METHOD M_StopCycle
mxStopCycle:= TRUE;
END_METHOD

METHOD M_StopDirect

IF mxCycleBusy THEN
	mxStopDirect:= TRUE;	
END_IF
END_METHOD

METHOD M_StopInit

IF mxInitBusy THEN 
	mxStopInit:= TRUE; 
END_IF
END_METHOD

ACTION Objects:

HydraulicCilinder(
	mxReset:= mxReset,
	mxEmergency:= mxEmergency, 
	mxAutoMode:= mxAutoMode, 
	EndPositionIn:= MachParameters.PositionUpStop,
	EndPositionOut:= ProdParameters.PositionDownStop,
	OffsetPosition:= MachParameters. PositionOffsetZero,
	OffsetAlarmPosition:= MachParameters.PositionOffsetAlarm,
	PositionPhysicalMeasured:=MachParameters.PositionPhyscialMeasured,
	PositionPhysicalMeasuredOld:=MachParameters.PositionPhysicalMeasuredOld,
	PhysicalOffsetPos:=MachParameters.PhysicalOffsetPos,
	RHSR_Blocked:=RHSR_Blocked,
	mxCycleBusy:=mxCycleBusy,
	mxInitBusy:=mxInitBusy,
	mxIsMovingIn=> mxCilIsMovingIn, 
	mxIsMovingOut=> mxCilIsMovingOut,
	ManSpeedCreepIn:=MachParameters.ManSpeedCreep,
	ManSpeedCreepOut:=MachParameters.ManSpeedCreep,
	ManSpeedSlowIn:=MachParameters.ManSpeedSlow,
	ManSpeedSlowOut:=MachParameters.ManSpeedSlow,
	ManSpeedIn:=MachParameters.ManSpeed,
	ManSpeedOut:=MachParameters.ManSpeed,
	mxIsIn=> mxCilIsIn, 
	mxIsOut=> mxCilIsOut,
	Errors=> Errors.HydraulicCilinder);
	
Vacuum(
	mxReset:= mxReset, 
	mxAutoMode:= mxAutoMode);

BlowOff(
	mxReset:= mxReset, 
	mxAutoMode:= mxAutoMode);
END_ACTION

END_FUNCTION_BLOCK

// ---- POUs/InMoldDrying/ProductForming/FB_ProductForming.TcPOU
FUNCTION_BLOCK FB_ProductForming
VAR CONSTANT
	sCycleStateTextDef: ARRAY[0..25]  OF STRING :=	
		['State 0: Wait for Start',
		'State 1: Start wire spray',
		'State 2: Move pond up',
		'State 3: Pond up, await pond up wait time',
		'State 4: Open pulp feeding valve and bubble valve',
		'State 5: Await feeding and bubble time',
		'State 6: Open the vacuum valve and await forming time',
		'State 7: Move pond down',
		'State 8: Start flash spray',
		'State 9: Start after vacuum time and await pre ignition time',
		'State 10: Await after vacuum time done',
		'State 11: Wait for transfer at down position',
		'State 12: Await after blow off time',
		'State 13: ',
		'State 14: ',
		'State 15: ',
		'State 16: ',
		'State 17: ',
		'State 18: ',
		'State 19: ',
		'State 20: Stop cycle state',
		'State 21: Stop direct state'
		];
	
	tCycleStateTimeouts: ARRAY[0..10] OF TIME := 
		[T#10S,T#10S,T#10S,T#10S,T#10S,T#10S,T#10S,T#10S,T#10S,T#10S,
		T#10S];

	sInitStateTextDef: ARRAY[0..10] OF STRING :=
		['State 0: Wait for Start',
		'State 1: Move machinepond down',
		'State 2: Move the spraybar to the rest position',
		'State 3: Description Init State 3',
		'State 4: Description Init State 4',
		'State 5: Description Init State 5',
		'State 6: Description Init State 6',
		'State 7: Description Init State 7',
		'State 8: Description Init State 8',
		'State 9: Description Init State 9',
		'State 10: Stop init state'];

	tInitStateTimeouts: ARRAY[0..10] OF TIME := 
		[T#10S,T#10S,T#10S,T#10S,T#10S,T#10S,T#10S,T#10S,T#10S,T#10S
		,T#10S];
END_VAR

VAR_INPUT
	mxResetCycleState				: BOOL;
	mxResetInitState				: BOOL;
	mxForceInit						: BOOL; (*Reset Calibration Flag*)
	mxReset							: BOOL;	(*Reset Error*)
	mxEmergency						: BOOL;
	mxAutoMode						: BOOL; (* TRUE = Automode *)
	mxStartCycle					: BOOL;
	mxEmptyMachine					: BOOL;
	mxFirstCycle					: BOOL;
	


	
	mxStartTransferMoldVacuum		: BOOL;

	mxAfterBlowOffIsOn				: BOOL;
	ActualPositionTransfermold		: REAL;
	TransfermoldDownPosition		: REAL; // Position at which the transfermold thinks its down.
	TransfermoldMovingDown			: BOOL; // Transfermold is moving down if true.
	TransfermoldMovingUp			: BOOL;
	RHSR_Blocked 					: BOOL;
	
	(*Signals*)
	sgTransferIsDown				: BOOL;(* Reset in cycle *)
	sgAtPosition					: BOOL;
	sgTransferToMoveUp				: BOOL;	
	SgTransferToDownForming			: BOOL; (* Reset at main cycle *)
	
END_VAR
VAR_IN_OUT
	MachParameters					: ST_ProductFormingMachPar;
	SysParameters					: ST_ProductFormingSysPar;
END_VAR
VAR_OUTPUT
(*Errors*)
	Errors							: ST_ProductFormingErrors;
	mxErrorInit						: BOOL;		(* Error, stop immediately. Initialisation neccesary *)
	mxErrorStopinPos				: BOOL;		(* Error, stop in position. Only reset neccesary *)

(* State vars *)
	mxCycleBusy						: BOOL;
	mxInitBusy						: BOOL;
	
(* Vars *)
	mxInitialized					: BOOL;

	mxCilIsMovingIn						: BOOL;
	mxCilIsMovingOut					: BOOL;
	mxCilIsIn							: BOOL;
	mxCilIsOut							: BOOL;

(*Signals*)	
	mxSprayBarAtRestPos					: BOOL;

	
END_VAR
VAR
(* State vars *)
	miCycleState					: INT :=0;
	miCycleOldstate					: INT :=0;
	mxCycleTransitionState			: BOOL := FALSE;
	sCycleStateText					: STRING;
	exCycleTimeOut					: BOOL;		(* Timeout for the whole programcycle *)
	CycleTimeout					: TON;
	CycleTimeOutUpFlank				: R_TRIG;
	mxCycleTimeoutEnable			: BOOL;
	CycleTime						: REAL;
	mxCycleHasError					: BOOL;
	miStopState						: INT;
	mxStopCycle						: BOOL;
	mxStopDirect					: BOOL;
	
	miInitState						: INT	:=0;
	miInitOldstate					: INT	:=0;
	mxInitTransitionState			: BOOL	:= FALSE;
	sInitStateText					: STRING;
	exInitTimeOut					: BOOL;		(* Timeout for the whole programcycle *)
	InitTimeout						: TON;
	InitTimeOutUpFlank				: R_TRIG;
	mxInitTimeoutEnable				: BOOL;
	InitTime						: REAL;
	mxInitHasError					: BOOL;
	mxStartInit						: BOOL;
	mxStopInit						: BOOL;
	
(* Objects *)
(* Forming Mold *)
	MoldVacuum						: FB_MonoValveNoFdbck;							
	MoldBlowOff						: FB_MonoValveNoFdbck;
(* MachinePond *)
	PondHydraulicCilinder			: FB_HydraulicCilinder;
	FeedingPulp						: FB_MonoValve2Fdbck;
(* SprayBar *)	
	WireSprayValve					: FB_MonoValveNoFdbck;
	FlashSprayValve					: FB_MonoValveNoFdbck;
	SprayBarMotor					: FB_NCAxis;	

	(* Interface signals pulp tanks, plup supply*)
	ixPulpTank01					AT %I*: BOOL;
	ixPulpTank02					AT %I*: BOOL;
	ixCssHasAnError					AT %I*: BOOL;
	
	TankLevel01						: FB_AnalogIn4_20mA;
	TankLevel02						: FB_AnalogIn4_20mA;
	
(* Vars *)

	T_PondUpWaitTime	: TON;
	T_FeedingPulp		: TON;
	T_Bubble			: TON;
	
	T_FirstVacuum		: TON;
	T_SecondVacuum		: TON;
	T_ThirdVacuum		: TON;

	T_FormingClosedTime : TON;

	
	FormingVacuumTime	: TIME;
	

	miWireSprayInterval	: INT;
	mxMoveForward		: BOOL;
	miFlashSprayInterval: INT;

	
	RT_ixPulpTank01		: R_TRIG;
	RT_ixPulpTank02		: R_TRIG;
	RT_FlashSprayStarted: R_TRIG;
	RT_InitBusy			: R_TRIG;

	mxPreIgnitionActive	: BOOL;

	mxSprayBarAtRestPosFront: BOOL;
	mxSprayBarAtRestPosBack: BOOL;
	T_SprayDelayTime	: TON;
	T_CycleTimeForKickoffs: TON;
	ActTimeSingleKO		: REAL;
	SR_TanksAreAllmostEmpty: SR;
	mxBubblingReady: BOOL;
	SR_CssHasError: SR;
END_VAR

Error();
Init();
Cycle();
Objects();

mxSprayBarAtRestPos:= mxSprayBarAtRestPosFront OR mxSprayBarAtRestPosBack;
	
mxSprayBarAtRestPosFront := ((SprayBarMotor.ActPosition <= MachParameters.SprayBar.PositionRestFront + 5) AND (SprayBarMotor.ActPosition >= MachParameters.SprayBar.PositionRestFront - 5));
mxSprayBarAtRestPosBack := ((SprayBarMotor.ActPosition <= MachParameters.SprayBar.PositionRestBack + 5) AND (SprayBarMotor.ActPosition >= MachParameters.SprayBar.PositionRestBack - 5));

ACTION Cycle:
(*StateChange (Transition)  Signalgeneration*)
mxCycleTransitionState:=(miCycleState<>miCycleOldstate);
(*State text*)
sCycleStateText:=sCycleStateTextDef[miCycleState];
(*Timeout Watchdog for Statemachine*)
mxCycleTimeoutEnable:=NOT (miCycleState=0) AND NOT mxReset;

CycleTimeout(IN:=mxCycleTimeoutEnable, PT:=tCycleStateTimeouts[miCycleState] );
CycleTimeOutUpFlank(CLK:=CycleTimeout.Q );
miCycleOldstate:=miCycleState;

(*Set Errorbit when Raising edge of Timeout has been detected*)
IF CycleTimeOutUpFlank.Q THEN
	exCycleTimeOut:=TRUE; 			(* 1 Timeout for the whole programcycle *)
END_IF

(*Function to reset the Statemachine*)
IF mxResetCycleState THEN
	mxResetCycleState:= FALSE;
	mxInitialized := FALSE;
	miCycleState:=0;
	miCycleOldstate:=miCycleState;
	mxCycleTransitionState:=FALSE;

	mxStartTransferMoldVacuum:= FALSE;
	mxAfterBlowOffIsOn := FALSE;
	mxStartCycle:= FALSE;
	mxStopCycle:= FALSE;
	mxStopDirect:=FALSE;

	T_FirstVacuum.In := FALSE;
	T_SecondVacuum.IN:= FALSE;
	T_ThirdVacuum.IN := TRUE;
	
	T_PondUpWaitTime.IN:= FALSE;
	T_FeedingPulp.IN:= FALSE;
	T_Bubble.IN:= FALSE;
	
	T_SprayDelayTime.IN:= FALSE;
	T_CycleTimeForKickoffs.IN := FALSE;
	SprayBarMotor.M_Stop();
	
	sgTransferIsDown := FALSE;
	sgAtPosition :=FALSE;
	sgTransferToMoveUp :=FALSE;	
	SgTransferToDownForming :=FALSE; 
END_IF

(*Definition State has Error*)
mxCycleHasError:=FALSE;


(* Set Forming vacuum time when switch over to next pulp tank,
Increase when flah spray is started*)
RT_ixPulpTank01(CLK:= ixPulpTank01);
RT_ixPulpTank02(CLK:= ixPulpTank02);
RT_InitBusy(CLK:= mxInitBusy);
RT_FlashSprayStarted(CLK:= miCycleState = 8);
	
IF RT_ixPulpTank01.Q OR RT_ixPulpTank02.Q OR RT_InitBusy.Q OR TRUE THEN // ----------------------------------------------------------------------------------- TRUE Weghalen wanneer wissel signaal actief
	FormingVacuumTime:= MachParameters.FormingMold.VacuumTime;
ELSIF RT_FlashSprayStarted.Q AND FALSE THEN								// ----------------------------------------------------------------------------------- IDEM voor false.
	IF ixPulpTank01 THEN
		FormingVacuumTime := FormingVacuumTime + (REAL_TO_TIME((TIME_TO_REAL(MachParameters.FormingMold.VacuumTimeIncr ) / 70.0) * (75 -  TankLevel01.EngUnits))); 
	ELSIF ixPulpTank02 THEN
		FormingVacuumTime := FormingVacuumTime + (REAL_TO_TIME((TIME_TO_REAL(MachParameters.FormingMold.VacuumTimeIncr ) / 70.0) * (75 -  TankLevel02.EngUnits))); 
	END_IF
END_IF


// 			Timers			//
T_FeedingPulp(IN:= , PT:= MachParameters.MachinePond.FeedingPulpTime); 
T_Bubble(IN:= , PT:= MachParameters.FormingMold.BubbleTime);
T_FormingClosedTime(IN:= , PT:= MachParameters.FormingMold.ClosedTime);
T_SprayDelayTime(IN:=, PT:=MachParameters.SprayBar.SprayDelayTime);
T_CycleTimeForKickoffs(IN:=, PT:=T#250S);
T_FirstVacuum(IN:= , PT:= FormingVacuumTime);
T_SecondVacuum(IN:= , PT:= MachParameters.FormingMold.SecondVacuum);
T_ThirdVacuum(IN:=, PT:=MachParameters.FormingMold.ThirdVacuum);

// Signal the transfermold that it can start moving down afet T2 has elapsed
IF T_SecondVacuum.Q THEN	
	T_SecondVacuum.IN:= FALSE;
	T_ThirdVacuum.IN := TRUE;
	SgTransferToDownForming:= TRUE; // send transfermold down
END_IF

IF T_ThirdVacuum.Q THEN
	T_ThirdVacuum.IN := FALSE;	
END_IF

// Close feeding pulp valve after timer is done
IF T_FeedingPulp.Q THEN 
	T_FeedingPulp.IN := FALSE;
	FeedingPulp.M_Close(); 
END_IF
			
(*Cycle State's*)
CASE miCycleState OF

{region "Steps overview"}	
	(*
	-Start wire spray
	-move pond up
	-Open blow off valve (bubble) 
	-Await bubble time
	-Close feeding valve/blow off valve/start vacuum + timer
	-Wait for vacuum timer
	-move pond down
	-Start flash spray
	-Start after vacuum timer/Pre-ignition timer
	-After vacuum time is done, -> Move down to Transfer Mold
	-Wait for transfer down 	<- from transfer mold
	-Open blow off valve
	-Start forming timer
	-Start blow off timer
	-Signal to transfer 		-> Move up to transfer mold
	-Wait for start forming (start cycle)		<- from transfer mold
	*)
{endregion}
	0:
		IF mxStopDirect THEN
			mxStopDirect:= FALSE;
			miCycleState:= 21;
		ELSIF mxStopCycle AND mxEmptyMachine THEN
			mxEmptyMachine:= FALSE;
			T_CycleTimeForKickoffs.IN := FALSE;	// Start timer to measure the cycle time of the transfer mold.
			miCycleState:= 0;
		ELSIF mxStopCycle THEN
			mxStopCycle:= FALSE;
			miStopState:= miCycleState;
			miCycleState:= 20;
		ELSIF mxStartCycle THEN
			mxStartCycle:= FALSE;
			T_CycleTimeForKickoffs.IN := TRUE;	// Start timer to measure the cycle time of the transfer mold.
			mxStartTransferMoldVacuum:= FALSE;
			
			mxMoveForward:= FALSE;				(* Check if at rest back position, then move forward, else move backward *)
			IF SprayBarMotor.ActPosition < MachParameters.SprayBar.PositionRestBack + 5 AND SprayBarMotor.ActPosition > MachParameters.SprayBar.PositionRestBack - 5 THEN
				mxMoveForward:= TRUE;
			END_IF	
			(* If parameter = 0 then do not perform spray, if 1 then always perform spray, other: perform every x time *)
			IF MachParameters.SprayBar.WireSprayInterval > 0 AND ((miWireSprayInterval = MachParameters.SprayBar.WireSprayInterval) OR MachParameters.SprayBar.WireSprayInterval = 1) THEN
				miWireSprayInterval:= miWireSprayInterval - 1;		
				miCycleState:= 1;
			ELSE
				miWireSprayInterval:= miWireSprayInterval - 1;
				miCycleState:=2 ;
			END_IF
			IF miWireSprayInterval <=0 THEN miWireSprayInterval:= MachParameters.SprayBar.WireSprayInterval; END_IF		//Write to par if is lower then 0
		END_IF
		
	
	1: // Start Wire Spray 
		IF mxMoveForward THEN
			IF SprayBarMotor.ActPosition >= MachParameters.SprayBar.PositionStartWireFwd THEN
				WireSprayValve.M_On();
			END_IF
			IF SprayBarMotor.ActPosition >= MachParameters.SprayBar.PositionStopWireFwd THEN
				WireSprayValve.M_Off();
			END_IF
		ELSE
			IF SprayBarMotor.ActPosition <= MachParameters.SprayBar.PositionStartWireBkw THEN
				WireSprayValve.M_On();
			END_IF
			IF SprayBarMotor.ActPosition <= MachParameters.SprayBar.PositionStopWireBkw THEN
				WireSprayValve.M_Off();
			END_IF
		END_IF
			
		IF mxStopDirect THEN
			mxStopDirect:= FALSE;
			miCycleState:= 21;
		ELSIF mxStopCycle THEN
			mxStopCycle:= FALSE;			
			miStopState:= miCycleState;
			miCycleState:= 20;
		ELSIF mxMoveForward  THEN
			IF SprayBarMotor.M_MoveAbsolute(Velocity:= MachParameters.SprayBar.AutoVelocity, Position:= MachParameters.SprayBar.PositionRestFront) THEN
				miCycleState:= 2;	
			END_IF
		ELSIF NOT mxMoveForward THEN
			IF SprayBarMotor.M_MoveAbsolute(Velocity:= MachParameters.SprayBar.AutoVelocity, Position:= MachParameters.SprayBar.PositionRestBack) THEN
				miCycleState:= 2;	
			END_IF
		END_IF
	
	2:	// Move pond up
		IF (PondHydraulicCilinder.ActPosition > (MachParameters.MachinePond.PositionUpStop - MachParameters.MachinePond.BubblingPositionOffset)) THEN
			IF MoldBlowOff.M_On() THEN T_Bubble.IN:= TRUE; END_IF  // When the machine pond is almost up -> Start bubbling (open valve)
		END_IF
	
		IF mxStopDirect THEN
			mxStopDirect:= FALSE;
			miCycleState:= 21;
		ELSIF mxStopCycle THEN
			mxStopCycle:= FALSE;
			PondHydraulicCilinder.M_Stop();		
			miStopState:= miCycleState;
			miCycleState:= 20;
		ELSIF PondHydraulicCilinder.M_Move(End_Position:= MachParameters.MachinePond.PositionUpStop, Slow_Position:= MachParameters.MachinePond.PositionUpSlow) THEN
			miCycleState:= 3;
		END_IF
	
	3:	// pulp supply open when bubbling is done.		
		IF mxStopDirect THEN
			mxStopDirect:= FALSE;
			miCycleState:= 21;
		ELSIF mxStopCycle THEN
			mxStopCycle:= FALSE;
			miStopState:= miCycleState;
			miCycleState:= 20;	
		ELSIF T_Bubble.Q OR TRUE THEN // REMOVE TRUE when done with testing.
			T_Bubble.IN := FALSE;
			MoldBlowOff.M_Off();	
		
			// open feeding valve
			FeedingPulp.M_Open();  
			T_FeedingPulp.IN:= TRUE;
			
			//Start first vacuum
			MoldVacuum.M_On();	// open the vacuum valve and start first vac. timer.
			T_FirstVacuum.IN := TRUE;	
			
			miCycleState:= 4;
		END_IF	
		
	4:	// First vacuum time is finished, start 2nd vacuum time	
		IF mxStopDirect THEN
			mxStopDirect:= FALSE;
			miCycleState:= 21;
		ELSIF mxStopCycle THEN
			mxStopCycle:= FALSE;
			miStopState:= miCycleState;
			miCycleState:= 20;	
		ELSIF T_FirstVacuum.Q THEN
			T_FirstVacuum.IN := FALSE;
			T_SecondVacuum.IN := TRUE;	
			miCycleState:= 5;
		END_IF		
	
	5:	///When first vacuum is finished and 2nd started, move pond down.
		IF mxStopDirect THEN
			mxStopDirect:= FALSE;
			miCycleState:= 21;
		ELSIF mxStopCycle THEN
			mxStopCycle:= FALSE;		
			miStopState:= miCycleState;
			miCycleState:= 20;
		ELSIF PondHydraulicCilinder.M_Move(End_Position:= MachParameters.MachinePond.PositionDownStop, Slow_Position:= MachParameters.MachinePond.PositionDownSlow) THEN
			T_SprayDelayTime.IN:= TRUE;		
			
			IF T_SprayDelayTime.Q THEN
				T_SprayDelayTime.IN :=FALSE;	
			
				mxMoveForward:= FALSE;
				IF SprayBarMotor.ActPosition < MachParameters.SprayBar.PositionRestBack + 5 AND SprayBarMotor.ActPosition > MachParameters.SprayBar.PositionRestBack - 5 THEN
					mxMoveForward:= TRUE;
				END_IF	
				
				(* If parameter = 0 then do not perform spray, if 1 then always perform spray, other: perform every x time *)
				IF MachParameters.SprayBar.FlashSprayInterval > 0 AND ((miFlashSprayInterval = MachParameters.SprayBar.FlashSprayInterval) OR MachParameters.SprayBar.FlashSprayInterval = 1) THEN
					miFlashSprayInterval:= miFlashSprayInterval - 1;
					miCycleState:= 6; 
				ELSE
					miFlashSprayInterval:= miFlashSprayInterval - 1;		
					miCycleState:= 7;
				END_IF
				IF miFlashSprayInterval <=0 THEN miFlashSprayInterval:= MachParameters.SprayBar.FlashSprayInterval; END_IF 	// Write to par if is lower then 0
			END_IF
		END_IF
	
	6: 	// Start flash spray 
		IF mxMoveForward THEN
			IF SprayBarMotor.ActPosition >= MachParameters.SprayBar.PositionStartFlashFwd THEN
				FlashSprayValve.M_On();
			END_IF
			IF SprayBarMotor.ActPosition >= MachParameters.SprayBar.PositionStopFlashFwd THEN
				FlashSprayValve.M_Off();
			END_IF
		ELSE
			IF SprayBarMotor.ActPosition <= MachParameters.SprayBar.PositionStartFlashBkw THEN
				FlashSprayValve.M_On();
			END_IF
			IF SprayBarMotor.ActPosition <= MachParameters.SprayBar.PositionStopFlashBkw THEN
				FlashSprayValve.M_Off();
			END_IF
		END_IF

		IF mxStopDirect THEN
			mxStopDirect:= FALSE;
			miCycleState:= 21;
		ELSIF mxStopCycle THEN
			mxStopCycle:= FALSE;
			miStopState:= miCycleState;
			miCycleState:= 20;
		ELSIF mxMoveForward THEN
			IF SprayBarMotor.M_MoveAbsolute(Velocity:= MachParameters.SprayBar.AutoVelocity, Position:= MachParameters.SprayBar.PositionRestFront) THEN
				miCycleState:= 7;	
			END_IF
		ELSIF NOT mxMoveForward THEN
			IF SprayBarMotor.M_MoveAbsolute(Velocity:= MachParameters.SprayBar.AutoVelocity, Position:= MachParameters.SprayBar.PositionRestBack) THEN
				miCycleState:= 7;	
			END_IF
		END_IF

	7:	// Close forming mold vacuum valve on the way down of transfermold.
		IF TransfermoldMovingDown AND (ActualPositionTransfermold < (TransfermoldDownPosition + MachParameters.FormingMold.StopVacuumAtTrPosOffset)) THEN
			T_ThirdVacuum.IN := FALSE; // Abort third vacuum timer, to indicate total time.				
			MoldVacuum.M_Off();
		END_IF
		
		IF TransfermoldMovingDown AND (ActualPositionTransfermold < (TransfermoldDownPosition + MachParameters.FormingMold.StartBlowOffAtTrPosOffset)) THEN				
			MoldBlowoff.M_On();
		END_IF

		IF mxStopDirect THEN
			mxStopDirect:= FALSE;
			miCycleState:= 21;
		ELSIF mxStopCycle THEN
			mxStopCycle:= FALSE;
			miStopState:= miCycleState;
			miCycleState:= 20;
		ELSIF sgTransferIsDown THEN
			sgTransferIsDown:= FALSE;
			miCycleState:= 8;
		END_IF
		
	8:	// Close time (time the transfer is closed on the formingmold).
		T_FormingClosedTime.IN:= TRUE;

		IF mxStopDirect THEN
			mxStopDirect:= FALSE;
			miCycleState:= 21;
		ELSIF mxStopCycle THEN
			mxStopCycle:= FALSE;
			miStopState:= miCycleState;
			miCycleState:= 20;
		ELSIF T_FormingClosedTime.Q THEN	// Signal main cycle that transfer to start moving up again.
			T_FormingClosedTime.In:= FALSE;
			sgTransferToMoveUp:=TRUE;
			miCycleState:= 9;
		END_IF

	
	9:	// Switch blowoff due to transfer position 
	//	IF TransfermoldMovingUp AND 
	//	(ActualPositionTransfermold > (TransfermoldDownPosition + MachParameters.FormingMold.StartBlowOffAtTrPosOffset)) THEN				
	//		MoldBlowoff.M_On();
	//	END_IF

		IF mxStopDirect THEN
			mxStopDirect:= FALSE;
			miCycleState:= 21;
		ELSIF mxStopCycle THEN
			mxStopCycle:= FALSE;
			miStopState:= miCycleState;
			miCycleState:= 20;
		ELSIF TransfermoldMovingUp AND 
		(ActualPositionTransfermold > (TransfermoldDownPosition + MachParameters.FormingMold.StopBlowOffAtTrPosOffset)) THEN				
			MoldBlowoff.M_Off();
			
			ActTimeSingleKO := TIME_TO_REAL(T_CycleTimeForKickOffs.ET);
			T_CycleTimeForKickoffs.IN := FALSE;
			miCycleState:= 0;
		END_IF
		
	(* Stop Cycle *)
	20:
		FeedingPulp.M_Close();				// on controlled stop, close the pulpfeeding valve to prevent flooding.
	
		IF mxStopDirect THEN
			mxStopDirect:= FALSE;
			miCycleState:= 21;
		ELSIF mxStartCycle THEN
			mxStartCycle:= FALSE;
			miCycleState:= miStopState;
			T_CycleTimeForKickoffs.IN := FALSE;	
		END_IF
	
	(* Stop Direct*)
	21:
		T_PondUpWaitTime.IN:= FALSE;
		T_FeedingPulp.IN:= FALSE;
		T_Bubble.IN:= FALSE;
		
		T_FirstVacuum.IN:= FALSE;
		T_SecondVacuum.IN:= FALSE;
		T_ThirdVacuum.IN := FALSE;
		
		T_CycleTimeForKickoffs.IN := FALSE;	// Start timer to measure the cycle time of the transfer mold.
		ActTimeSingleKO := 0;
		
	(* Forming Mold *)
		MoldVacuum.M_Off();				
		MoldBlowOff.M_Off();
	(* MachinePond *)
		PondHydraulicCilinder.M_StopDirect();
		FeedingPulp.M_Close();
	(* SprayBar *)	
		WireSprayValve.M_Off();
		FlashSprayValve.M_Off();
		SprayBarMotor.M_Stop();

		mxStartCycle:= FALSE;
		mxStopCycle:= FALSE;
		mxStopDirect:=FALSE;
		mxInitialized:= FALSE;

		sgTransferIsDown := FALSE;
		sgAtPosition :=FALSE;
		sgTransferToMoveUp :=FALSE;	
		SgTransferToDownForming :=FALSE; 
		
		miCycleState:= 0;

END_CASE

mxCycleBusy:= miCycleState<>0 AND NOT (miCycleState=20);
END_ACTION

ACTION Error:
SR_TanksAreAllmostEmpty(SET1:=(TankLevel01.EngUnits < 5) AND (TankLevel02.EngUnits < 5), RESET:=mxReset, Q1=>Errors.LowLvlOnBothTanks);  
SR_CssHasError(SET1:=ixCssHasAnError, Reset:=mxReset, Q1=>Errors.CssHasError);



(*************************************************************************************************)
mxErrorInit:= Errors.HydraulicPump.Thermal;
mxErrorStopinPos:= FALSE;
END_ACTION

ACTION Init:
(*StateChange (Transition)  Signalgeneration*)
mxInitTransitionState:=(miInitState<>miInitOldstate);
(*State text*)
sInitStateText:=sInitStateTextDef[miInitState];
(*Timeout Watchdog for Statemachine*)
mxInitTimeoutEnable:=NOT (miInitState=0)  AND NOT mxReset;

InitTimeout(IN:=mxInitTimeoutEnable  , PT:=tInitStateTimeouts[miInitState] );
InitTimeOutUpFlank(CLK:=InitTimeout.Q );
miInitOldstate:=miInitState;

(*Set Errorbit when Raising edge of Timeout has been detected*)
IF InitTimeOutUpFlank.Q THEN
	exInitTimeOut:=TRUE; 			(* 1 Timeout for the whole programcycle *)
END_IF

(*Function to reset the Statemachine*)
IF mxResetInitState THEN
	mxResetInitState:=FALSE;
	mxInitialized:= FALSE;
	miInitState:=0;
	miInitOldstate:=miInitState;
	mxInitTransitionState:=FALSE;
	
	mxStartInit:= FALSE;
	mxStopInit:= FALSE;
END_IF

(*Definition State has Error*)
mxInitHasError:=FALSE;

CASE miInitState OF
	0:
		IF mxStartInit THEN
			mxStartInit:= FALSE;
			mxInitialized:= FALSE;

		(* Forming Mold *)
			MoldVacuum.M_Off();				
			MoldBlowOff.M_Off();
		(* MachinePond *)
			FeedingPulp.M_Close();
		(* SprayBar *)	
			WireSprayValve.M_Off();
			FlashSprayValve.M_Off();
			(* AT init write intervals *)
			miWireSprayInterval:= MachParameters.SprayBar.WireSprayInterval;
			miFlashSprayInterval:= MachParameters.SprayBar.FlashSprayInterval;
			
			miInitState:= 1;
		END_IF

	(* Move Pond down *)	
	1:
		IF mxStopInit THEN
			mxStopInit:= FALSE;
			
			miInitState:= 10;			
		ELSIF PondHydraulicCilinder.M_Move(End_Position:= MachParameters.MachinePond.PositionDownStop, Slow_Position:= MachParameters.MachinePond.PositionDownSlow) THEN
			
			miInitState:= 2;
		END_IF				

	(* Move spraybar to rest position *)	
	2:
		IF mxStopInit THEN
			mxStopInit:= FALSE;
			
			miInitState:= 10;			
		ELSIF SprayBarMotor.M_MoveAbsolute(Position:= MachParameters.SprayBar.PositionRestBack, Velocity:= MachParameters.SprayBar.AutoVelocity) THEN
			mxInitialized:= TRUE;
			
			// stop the pump en cylinder of the pond
			PondHydraulicCilinder.M_Stop();
			
			miInitState:= 0;
		END_IF

	10:
		PondHydraulicCilinder.M_Stop();
		SprayBarMotor.M_Stop();

		mxStartInit:= FALSE;
		mxStopInit:= FALSE;
		mxInitialized:= FALSE;
		
		miInitState:= 0;
END_CASE

mxInitBusy:= miInitState<>0;
END_ACTION

METHOD M_EmptyMachine

IF mxCycleBusy THEN
	mxEmptyMachine:= TRUE;	
END_IF
END_METHOD

METHOD M_StartCycle

IF NOT mxCycleBusy THEN
	mxStartCycle:= TRUE;
	mxStopCycle:=False;
END_IF
END_METHOD

METHOD M_StartInit

IF NOT mxInitBusy THEN 
	mxStartInit:= TRUE;
END_IF
END_METHOD

METHOD M_StopCycle

IF mxCycleBusy THEN
	mxStopCycle:= TRUE;
END_IF
END_METHOD

METHOD M_StopDirect

IF mxCycleBusy THEN
	mxStopDirect:= TRUE;	
END_IF
END_METHOD

METHOD M_StopInit

IF mxInitBusy THEN 
	mxStopInit:= TRUE; 
END_IF
END_METHOD

ACTION Objects:

MoldVacuum(
	mxReset:= mxReset,
	mxAutoMode:= mxAutoMode,
	mxEmergency:= mxEmergency);

MoldBlowOff(
	mxReset:= mxReset,
	mxAutoMode:= mxAutoMode,
	mxEmergency:= mxEmergency);
	
PondHydraulicCilinder(
	mxReset:= mxReset,
	mxAutoMode:= mxAutoMode,
	mxEmergency:= mxEmergency,
	EndPositionIn:= MachParameters.MachinePond.PositionDownStop,
	EndPositionOut:= MachParameters.MachinePond.PositionUpStop,
	OffsetPosition:= MachParameters.MachinePond.PositionOffsetZero,
	OffsetAlarmPosition:= MachParameters.MachinePond.PositionOffsetAlarm,
	PositionPhysicalMeasured:=MachParameters.MachinePond.PositionPhyscialMeasured,
	PositionPhysicalMeasuredOld:=MachParameters.MachinePond.PositionPhysicalMeasuredOld,
	PhysicalOffsetPos:=MachParameters.MachinePond.PhysicalOffsetPos,
	RHSR_Blocked := RHSR_Blocked,
	SlowValveIsInverted := FALSE,
	mxIsVertical := TRUE,
	mxIsMovingIn=> mxCilIsMovingIn, 
	mxIsMovingOut=> mxCilIsMovingOut, 
	mxIsIn=> mxCilIsIn, 
	mxIsOut=> mxCilIsOut,
	Errors=> );


FeedingPulp(
	mxReset:= mxReset,
	mxAutoMode:= mxAutoMode,
	mxEmergency:= mxEmergency,
	MachParameters:= MachParameters.MachinePond.FeedingPulp);

WireSprayValve(
	mxReset:= mxReset,
	mxAutoMode:= mxAutoMode,
	mxEmergency:= mxEmergency);

FlashSprayValve(
	mxReset:= mxReset,
	mxAutoMode:= mxAutoMode,
	mxEmergency:= mxEmergency);

SprayBarMotor(
	mxEnable:= NOT mxEmergency, 
	mxInhibit:=FALSE , 
	mxAutoMode:= mxAutoMode, 
	mxReset:= mxreset, 
	mxEmergency:= mxEmergency, 
	mxSimulation:= , 
	mxFirstCycle:= mxFirstCycle, 
	mxResetCycle:= , 
	mxDisable_Positive:=FALSE , 
	mxDisable_Negative:=FALSE , 
	mxBlockHMI:=FALSE , 
	mrOverride:= 100,
	mrHomePos:=MachParameters.SprayBar.PositionHome,
	mrVelocityManual:= MachParameters.SprayBar.ManualVelocity, 
	SysParameters:= SysParameters.SprayBar, 
	mxCycleBusy=> , 
	mxRunning=> , 
	Errors=> errors.SprayBar.NCAxisError, 
	Error=> , 
	ErrorStop=> , 
	axStatus=> , 
	ActPosition=> , 
	ActVelocity=> , 
	axAxis=> );
	
TankLevel01(
	EngLowLimit:= 0, 
	EngUpperLimit:= 100, 
	maOut=> , 
	EngUnits=> , 
	EngFilt=> , 
	OverRange=> , 
	UnderRange=> );
	
TankLevel02(
	EngLowLimit:= 0, 
	EngUpperLimit:= 100, 
	maOut=> , 
	EngUnits=> , 
	EngFilt=> , 
	OverRange=> , 
	UnderRange=> );
END_ACTION

END_FUNCTION_BLOCK

// ---- POUs/Standard/HydraulicCilinder/FB_HydraulicCilinder.TcPOU
FUNCTION_BLOCK FB_HydraulicCilinder

VAR_INPUT

	mxReset							: BOOL;	(*Reset Error*)
	mxEmergency						: BOOL;
	mxAutoMode						: BOOL; (* TRUE = Automode *)
	EndPositionIn					: REAL;
	EndPositionOut					: REAL;
	OffsetPosition					: REAL;
	OffsetAlarmPosition				: REAL;	
	PositionPhysicalMeasured		: REAL;	
	RHSR_Blocked					: BOOL; (*IF true, then movement of the cylinder is blocked by the red hot safetyrules.*)
	SlowValveIsInverted				: BOOL;
	mxIsVertical					: BOOL;
	
		// used in M_move
	mxMoveIn						: BOOL;
	mxMoveOut						: BOOL;
	
END_VAR
VAR_OUTPUT
(*Errors*)
	Errors							: ST_HydraulicErrors;
	mxErrorInit						: BOOL;		(* Error, stop immediately. Initialisation neccesary *)
	mxErrorStopinPos				: BOOL;		(* Error, stop in position. Only reset neccesary *)

(* State vars *)
	mxCycleBusy						: BOOL;
	mxInitBusy						: BOOL;
	
(* Vars *)
	mxInitialized					: BOOL;
	ActPosition						: REAL;
	ActMeasuredPosition				: REAL;
	mxSlowActive					: BOOL;
	mxIsMovingIn					: BOOL;
	mxIsMovingOut					: BOOL;
	mxIsIn							: BOOL;
	mxIsOut							: BOOL;
END_VAR
VAR
(* State vars *)
	miCycleState					: INT :=0;
	miCycleOldstate					: INT :=0;
	mxCycleTransitionState			: BOOL := FALSE;
	sCycleStateText					: STRING;
	exCycleTimeOut					: BOOL;		(* Timeout for the whole programcycle *)
	CycleTimeout					: TON;
	CycleTimeOutUpFlank				: R_TRIG;
	mxCycleTimeoutEnable			: BOOL;
	CycleTime						: REAL;
	mxCycleHasError					: BOOL;
	miStopState						: INT;
	mxStartCycle					: BOOL;
	mxStopCycle						: BOOL;
	mxStopDirect					: BOOL;
	
	miInitState						: INT	:=0;
	miInitOldstate					: INT	:=0;
	mxInitTransitionState			: BOOL	:= FALSE;
	sInitStateText					: STRING;
	exInitTimeOut					: BOOL;		(* Timeout for the whole programcycle *)
	InitTimeout						: TON;
	InitTimeOutUpFlank				: R_TRIG;
	mxInitTimeoutEnable				: BOOL;
	InitTime						: REAL;
	mxInitHasError					: BOOL;
	mxStartInit						: BOOL;
	mxStopInit						: BOOL;

	(* Objects *)
	HydraulicIn						: FB_MonoValveNoFdbck;
	HydraulicOut					: FB_MonoValveNoFdbck;
	HydraulicSlow					: FB_MonoValveNoFdbck;
	HydraulicPos 					: FB_BalluffPosition;

	RodSidePressure					: FB_AnalogIn4_20mA;
	BottomSidePressure				: FB_AnalogIn4_20mA;
	
	EndPosition						: REAL; (* Destination position *)
	SlowPosition					: REAL; (* Slow position *)

	FT_ValveInOff					: F_TRIG;
	FT_ValveOutOff					: F_TRIG;
	HydraulicStoredPosition			: REAL;
	

	
	Hysteresis: REAL := 1;
	mxMoveReadyWithoutMoving: BOOL;
	
	RT_Emergency: R_Trig;
	FT_AutoMode: F_TRIG;
END_VAR
VAR_IN_OUT
	PositionPhysicalMeasuredOld		: REAL;
	PhysicalOffsetPos				: REAL;
END_VAR

Error();
Objects();

RT_Emergency(CLK:= mxEmergency);
FT_AutoMode(CLK:=mxAutoMode);

Hysteresis := 3;

// Calculate correction on actual balluf position to a virtual "zero" position.
IF PositionPhysicalMeasured <> PositionPhysicalMeasuredOld THEN
	PhysicalOffsetPos := (HydraulicPos.Position- (OffsetPosition + PositionPhysicalMeasured));
END_IF

// Create a virtual zero position by substracting a calculated offset
ActPosition:= HydraulicPos.Position - PhysicalOffsetPos;
ActMeasuredPosition:= HydraulicPos.Position;

mxIsMovingIn:= HydraulicIn.mxIsOn;
mxIsMovingOut:= HydraulicOut.mxIsOn;

mxIsIn:= (ActPosition <= (EndPositionIn + Hysteresis)) AND (ActPosition >= (EndPositionIn - Hysteresis));
mxIsOut:= (ActPosition <= (EndPositionOut + Hysteresis)) AND (ActPosition >= (EndPositionOut - Hysteresis));

(*Overwrite previous value*)
PositionPhysicalMeasuredOld := PositionPhysicalMeasured;

(* Used for sending slow settings to flow/pressure *) 
mxSlowActive:= HydraulicSlow.mxIsOn;


// Close valves on emergency stop.
IF RT_Emergency.Q OR FT_AutoMode.Q THEN
	HydraulicSlow.M_Off();
	HydraulicIn.M_Off();
	HydraulicOut.M_Off();
END_IF

ACTION Error:
Errors.BallufError:= HydraulicPos.Error;

(* When out of range up/down position *)

	IF (mxIsVertical AND (ActPosition > (EndPositionIn + OffsetAlarmPosition) OR ActPosition < (EndPositionOut - OffsetAlarmPosition))) OR 
		(NOT mxIsVertical AND (ActPosition < (EndPositionIn - OffsetAlarmPosition) OR ActPosition > (EndPositionOut + OffsetAlarmPosition))) THEN
		Errors.PositionError:= TRUE;
	ELSIF mxReset THEN
		Errors.PositionError:= FALSE;
	END_IF

(* Als valve up/down uit gaat, positie opslaan en controleren of deze veranderd tov de act positie*)
FT_ValveInOff(CLK:= HydraulicIn.mxIsOn);
FT_ValveOutOff(CLK:= HydraulicOut.mxIsOn);
IF FT_ValveInOff.Q OR FT_ValveOutOff.Q THEN HydraulicStoredPosition:= ActPosition; END_IF
IF mxReset THEN
	HydraulicStoredPosition:= ActPosition;
	Errors.IsMovingWithoutActivation:= FALSE;
ELSIF NOT HydraulicIn.mxIsOn AND NOT HydraulicOut.mxIsOn AND ((HydraulicStoredPosition > (ActPosition + 10)) OR (HydraulicStoredPosition < (ActPosition - 10))) THEN
	Errors.IsMovingWithoutActivation:= TRUE;
END_IF

(***************************************************************************************)
mxErrorStopInPos:= Errors.PositionError OR Errors.IsMovingWithoutActivation;
mxErrorInit:= FALSE;
END_ACTION

METHOD M_Move : BOOL
VAR_INPUT
	End_Position		: REAL; (* Destination position *)
	Slow_Position		: REAL; (* Slow position *)
END_VAR
VAR_OUTPUT
END_VAR
VAR


	mxMoveINReady: BOOL;
	mxMoveOutReady: BOOL;


END_VAR
(* Pass through parameters *) 
EndPosition:= End_Position;
SlowPosition:= Slow_Position;


mxMoveReadyWithoutMoving := FALSE;

(* bv atc pos = 0, end = 100  *)
IF (mxIsVertical AND (ActPosition <= (EndPosition - Hysteresis)) AND NOT mxMoveOut) OR			// Vertical movement (up)
	(NOT mxIsVertical AND (ActPosition >= (EndPosition + Hysteresis))  AND NOT mxMoveOut) THEN		// Horizontal movement (in)
	mxMoveIn:= TRUE;
	MxMoveOut:= FALSE;
	HydraulicIn.M_On();
	HydraulicOut.M_Off(); 	
ELSIF (mxIsVertical AND (ActPosition >= (EndPosition + Hysteresis)) AND NOT mxMoveIn) OR 			// Vertical movement (down)
	(NOT mxIsVertical AND (ActPosition <= (EndPosition - Hysteresis)) AND NOT mxMoveIn) THEN		// Horizontal movement (out)
	mxMoveIn:= FALSE;
	MxMoveOut:= TRUE;
	HydraulicIn.M_Off();
	HydraulicOut.M_On(); 
ELSE
	mxMoveReadyWithoutMoving:=TRUE;
END_IF

(* Move in *)	
IF mxMoveIn THEN
	IF (mxIsVertical AND (ActPosition > SlowPosition)) OR 				// Vertical movement
		(NOT mxIsVertical AND (ActPosition < SlowPosition))	THEN 		// Horizontal movement.
		HydraulicSlow.M_On();
	END_IF
END_IF

(* Move out *)
IF mxMoveOut THEN
	IF (mxIsVertical AND (ActPosition < SlowPosition)) OR 				// Vertical movement
	(NOT mxIsVertical AND (ActPosition > SlowPosition)) THEN			// Horizontal movement
		HydraulicSlow.M_On();
	END_IF
END_IF

mxMoveInReady := (mxMoveIn AND ((ActPosition >= (EndPosition - Hysteresis)) AND (ActPosition <= (EndPosition + Hysteresis))));
mxMoveOutReady := (mxMoveOut AND ((ActPosition >= (EndPosition - Hysteresis)) AND (ActPosition <= (EndPosition + Hysteresis))));			

// reset directional bits to zero when leaving this method.
IF mxMoveInReady OR mxMoveOutReady OR mxMoveReadyWithoutMoving THEN
	mxMoveIn:= FALSE;
	MxMoveOut:= FALSE;
	
	HydraulicIn.M_Off();
	HydraulicOut.M_Off();
	HydraulicSlow.M_Off();
END_IF

M_MOVE := mxMoveInReady OR mxMoveOutReady OR mxMoveReadyWithoutMoving;
END_METHOD

METHOD M_Stop : BOOL;
HydraulicIn.M_Off();
HydraulicOut.M_Off();
HydraulicSlow.M_Off();

mxMoveIn := FALSE;
mxMoveOut := FALSE;

M_Stop:= TRUE;
END_METHOD

METHOD M_StopDirect

HydraulicIn.M_Off();
HydraulicOut.M_Off();
HydraulicSlow.M_Off();
END_METHOD

ACTION Objects:
(* Objects Call *)
BottomSidePressure(
	EngLowLimit:=0, 
	EngUpperLimit:=315, 
	maOut=> , 
	EngUnits=> , 
	EngFilt=> , 
	OverRange=> , 
	UnderRange=> );

RodSidePressure(
	EngLowLimit:=0, 
	EngUpperLimit:=315, 
	maOut=> , 
	EngUnits=> , 
	EngFilt=> ,
	OverRange=> ,
	UnderRange=> );

HydraulicIn(
	mxReset:= mxReset, 
	mxEmergency:= mxEmergency, 
	mxAutoMode:= mxAutoMode,
	RHSR_Blocked := RHSR_Blocked);

HydraulicOut(
	mxReset:= mxReset, 
	mxEmergency:= mxEmergency, 
	mxAutoMode:= mxAutoMode,
 	RHSR_Blocked:=RHSR_Blocked);

HydraulicSlow(
	mxReset:= mxReset, 
	mxEmergency:= mxEmergency, 
	mxAutoMode:= mxAutoMode,
	SlowValveIsInverted := SlowValveIsInverted,
	RHSR_Blocked:=RHSR_Blocked);

HydraulicPos();
END_ACTION

END_FUNCTION_BLOCK

// ---- POUs/Standard/Valves/FB_MonoValve2Fdbck.TcPOU
FUNCTION_BLOCK FB_MonoValve2Fdbck
VAR_INPUT
	mxReset						: BOOL;	(*Reset Error*)
	mxEmergency					: BOOL;
	mxAutoMode					: BOOL; (* TRUE = Automode *)
	mxCheckCilinder				: BOOL:= TRUE;
END_VAR
VAR_IN_OUT
	MachParameters					: ST_CilinderParameters;
END_VAR
VAR_OUTPUT
	mxIsIn						: BOOL;
	mxIsOut						: BOOL;
	mxIsOpen					: BOOL;
	mxIsClosed					: BOOL;
	Errors						: ST_CilinderErrors;
	
	mxErrorInit: BOOL;
	mxErrorStopInPos: BOOL;

END_VAR
VAR
	Check						: FB_CheckCilinder;
	
	QxIn	 					AT %Q*: BOOL;
	QxOut						AT %Q*: BOOL;
	IxIsIn						AT %I*: BOOL;
	IxIsOut						AT %I*: BOOL;

	mxHMI_In					: BOOL;
	mxHMI_Out					: BOOL;
	mxHMI_Open					: BOOL;
	mxHMI_Close					: BOOL;
	RT_HMI_In					: R_TRIG;
	RT_HMI_Out					: R_TRIG;
END_VAR

Error();

RT_HMI_In(CLK:= NOT mxAutoMode AND (mxHMI_In OR mxHMI_Open));
RT_HMI_Out(CLK:= NOT mxAutoMode AND (mxHMI_Out OR mxHMI_Close));

(* Manual *)
IF RT_HMI_In.Q THEN M_In(); END_IF
IF RT_HMI_Out.Q THEN M_Out(); END_IF

(* Reset Outputs *)

//IF IxIsIn THEN QxIn:= FALSE; END_IF
//IF IxIsOut THEN QxOut:= FALSE; END_IF

(* Status *)
mxIsIn:= mxIsOpen:= IxIsIn;
mxIsOut:= mxIsClosed:= IxIsOut;

ACTION Error:
Check(
	MoveCilOut:= qxOut,
	MoveCilin:= qxIn,
	CheckCilinder:= mxCheckCilinder,
	SensorOut:=  mxIsOut OR mxIsClosed, // mx closed and open omgedraaid (20180528 -> Bateu*)
	SensorIn:= mxIsIn OR mxIsOpen,
	TimMax:= MachParameters.T_GuardTimeError,
	mxReset:= mxReset,
	ErrorCilinder=> Errors.Cilinder,
	ErrorCilinderOut=> ,
	ErrorCilinderIn=> ,
	ErrorEndNotReached=> ,
	ErrorSensorSwitched=> ,
	Time_Cil_Out=> ,
	Time_Cil_In=> );

(* Too slow errors, only messages *)
Errors.CilinderSlow_IN	:=	mxCheckCilinder AND (Check.Time_Cil_In > MachParameters.T_GuardTimeWarning_IN);
Errors.CilinderSlow_OUT	:=	mxCheckCilinder AND (Check.Time_Cil_Out > MachParameters.T_GuardTimeWarning_OUT);

(**********************************************************************************************************)
mxErrorStopinPos:= FALSE;
mxErrorInit:= Errors.Cilinder;
END_ACTION

METHOD PUBLIC M_Close: BOOL
VAR_INPUT
END_VAR
QxIn:= FALSE;

(* Return value *)
M_Close:= IxIsOut;
END_METHOD

METHOD PUBLIC M_In : BOOL
VAR_INPUT
END_VAR

QxIn:= TRUE;


(* Return value *)
M_In:= IxIsIn;
END_METHOD

METHOD PUBLIC M_Open : BOOL
VAR_INPUT
END_VAR

QxIn:= TRUE;


(* Return value *)
M_Open:= IxIsIn;
END_METHOD

METHOD PUBLIC M_Out: BOOL
VAR_INPUT
END_VAR
QxIn:= FALSE;

(* Return value *)
M_Out:= IxIsOut;
END_METHOD

END_FUNCTION_BLOCK

// ---- POUs/InMoldDrying/HydrolicsMain/FB_HydraulicsMain.TcPOU
FUNCTION_BLOCK FB_HydraulicsMain
VAR CONSTANT
	sCycleStateTextDef: ARRAY[0..20]  OF STRING :=	
		['State 0: Wait for Start',
		'State 1: Check Oil temperature and oil levels and Check all valves are in de-energised state',
		'State 2: When pump is running start the cooler and filterpump',
		'State 3: When pumps are running open circulation valve',
		'State 4: Check ciruclation valve is open, open Accumlator valve',
		'State 5: Check if Accu valve is open, and wait 15s',
		'State 6: Open the blocking valve',
		'State 7: Check if the blocking valve is open, and if pressure > x',
		'State 8: Main Hydraulics running',
		'State 9: Check if all analog valves are in the safe state',
		'State 10: Close presurize pumpvalve, stop cooling fan and filtermotor',
		'State 11: Close blocking valve and stop pump',
		'State 12: Spare',
		'State 13: [Paused: Close blocking valve]',
		'State 14: [Paused: Awaiting Restart]',
		'State 15: [Stopped Direct]'];
	
	tCycleStateTimeouts: ARRAY[0..10] OF TIME := 
		[T#10S,T#10S,T#10S,T#10S,T#10S,T#10S,T#10S,T#10S,T#10S,T#10S,
		T#10S];

	sInitStateTextDef: ARRAY[0..10] OF STRING :=
		['State 0: Wait for Init Start',
		'State 1: Await pressure relief',
		'State 2: Move up',
		'State 3: Description Init State 3',
		'State 4: Description Init State 4',
		'State 5: Description Init State 5',
		'State 6: Description Init State 6',
		'State 7: Description Init State 7',
		'State 8: Description Init State 8',
		'State 9: Description Init State 9',
		'State 10: Stop init state'];

	tInitStateTimeouts: ARRAY[0..10] OF TIME := 
		[T#10S,T#10S,T#10S,T#10S,T#10S,T#10S,T#10S,T#10S,T#10S,T#10S
		,T#10S];
END_VAR
VAR_INPUT
	mxReset								: BOOL;	(*Reset Error*)
	mxEmergency							: BOOL; // Used when a emergency stop button was pushed.
	mxDoorOpened						: BOOL;	// Used when a door was opened in the system
	mxAutoMode							: BOOL; (* TRUE = Automode *)
	PlcCycleTime						: REAL;
	
	
	
	(*State vars*)
	mxResetCycleState					: BOOL;
	mxResetInitState					: BOOL;
END_VAR
VAR_IN_OUT
	MachineParameters					: ST_HydraulicsMainMachPar;
END_VAR
VAR_OUTPUT
(*Errors*)
	Errors								: ST_HydraulicsMainErrors;
	mxErrorInit							: BOOL;		(* Error, stop immediately. Initialisation neccesary *)
	mxErrorStopinPos					: BOOL;		(* Error, stop in position. Only reset neccesary *)
	
	(* State vars *)
	mxCycleBusy							: BOOL;
	mxInitbusy							: BOOL;
	mxCycleInPause						: BOOL;
(* Vars *)
	mxInitialized						: BOOL;
	
	mxHydraulicsReady					: BOOL;
END_VAR
VAR
	(* State vars *)
	miCycleState					: INT :=0;
	miCycleOldstate					: INT :=0;
	mxCycleTransitionState			: BOOL := FALSE;
	sCycleStateText					: STRING;
	exCycleTimeOut					: BOOL;		(* Timeout for the whole programcycle *)
	CycleTimeout					: TON;
	CycleTimeOutUpFlank				: R_TRIG;
	mxCycleTimeoutEnable			: BOOL;
	CycleTime						: REAL;
	mxCycleHasError					: BOOL;
	miStopState						: INT;
	mxStartCycle					: BOOL;
	mxStopCycle						: BOOL;
	mxStopDirect					: BOOL;
	mxStopCycleEmpty				: BOOL;
	
	miInitState						: INT	:=0;
	miInitOldstate					: INT	:=0;
	mxInitTransitionState			: BOOL	:= FALSE;
	sInitStateText					: STRING;
	exInitTimeOut					: BOOL;		(* Timeout for the whole programcycle *)
	InitTimeout						: TON;
	InitTimeOutUpFlank				: R_TRIG;
	mxInitTimeoutEnable				: BOOL;
	InitTime						: REAL;
	mxInitHasError					: BOOL;
	mxStartInit						: BOOL;
	mxStopInit						: BOOL;	

	ixHydraulicsMcc24vError				AT %I*: BOOL;
	ixCabinetCoolerError				At %I*: BOOL;
	
	ixTemperatureSwitch40c				AT %I*: BOOL;
	ixTemperatureSwitch55c				AT %I*: BOOL;
	ixTemperatureSwitchTooHigh			AT %I*: BOOL;
	
	ixPressureFilterAt75				AT %I*: BOOL;
	ixPressureFilterAt100				AT %I*: BOOL;
	
	ixAuxFilterAt75						AT %I*: BOOL;
	ixAuxFilterAt100					AT %I*: BOOL;
	
	ixOilLvlTooLow						AT %I*: BOOL;
	ixOilLvlLow							AT %I*: BOOL;
	
	FT_AutoMode							: F_TRIG;
	
	(* Objects *)
	HydraulicPump						: FB_MotorSS;
	FilterMotor							: FB_Motor;
	CoolingFan							: FB_Motor;
	
	PressurizePumpValve					: FB_MonoValveNoFdbck;
	AccuDrainValve						: FB_MonoValveNoFdbck;
	IsolationValve						: FB_MonoValveNoFdbck;
	
	OilTemperature						: FB_AnalogIn4_20mA;
	MainSystemPressure					: FB_AnalogIn4_20mA;
	
	HmiForceCool						: BOOL;
	FT_ForceCool						: F_TRIG;
	T_DelayOpenBlockingValve			: TON;
	SR_TempTooHigh						: SR;
	SR_LevelTooLow						: SR;
	SR_Filter100Dirty					: SR;
	SR_AuxFilter100Dirty				: SR;
	SR_Filter75DirtyWarning				: SR;
	SR_AuxFilter75DirtyWarning			: SR;

	SR_CabinetCoolerError				: SR;
	SR_HydraulicsMcc24VError			: SR;
	RT_Doorsopenend						: R_TRIG;	// Used to produce a situation that is safe when doors are openend, but is also quick in restarting the machine
	
	mxTest1								: BOOL;
	T_DepresurizePump					: TON;
	RT_OilCoolerOn						: R_TRIG;
	FT_OilCoolerOff						: F_TRIG;
	FT_Emergency						: F_Trig;
	
	mxTest5: BOOL;
	RT_EmergencyStop: R_TRIG;

END_VAR

Cycle();
Error();
Objects();

// If both emergencies become zero, recheck if cooler needs to run.
FT_Emergency(CLK:=mxEmergency OR mxDoorOpened);
RT_OilCoolerOn(CLK:=ixTemperatureSwitch55c);
FT_OilCoolerOff (CLK:=ixTemperatureSwitch40c);

IF ((RT_OilCoolerOn.q) OR (FT_Emergency.Q AND ixTemperatureSwitch55c)) AND NOT CoolingFan.IsRunning THEN
	CoolingFan.M_Start();
END_IF

IF FT_OilCoolerOff.q AND CoolingFan.IsRunning THEN
	CoolingFan.M_Stop();
END_IF

ACTION Cycle:
(*StateChange (Transition)  Signalgeneration*)
mxCycleTransitionState:=(miCycleState<>miCycleOldstate);
(*State text*)
sCycleStateText:=sCycleStateTextDef[miCycleState];
(*Timeout Watchdog for Statemachine*)
mxCycleTimeoutEnable:=NOT (miCycleState=0) AND NOT mxReset;

CycleTimeout(IN:=mxCycleTimeoutEnable  , PT:=tCycleStateTimeouts[miCycleState] );
CycleTimeOutUpFlank(CLK:=CycleTimeout.Q );
miCycleOldstate:=miCycleState;

(*Set Errorbit when Raising edge of Timeout has been detected*)
IF CycleTimeOutUpFlank.Q THEN
	exCycleTimeOut:=TRUE; 			(* 1 Timeout for the whole programcycle *)
END_IF

(*Function to reset the Statemachine*)
IF mxResetCycleState THEN
	mxResetCycleState:= FALSE;
	mxInitialized := FALSE;
		
	miCycleState:=0;
	mxCycleTransitionState:=FALSE;

	mxStartCycle:= FALSE;
	mxStopCycle:= FALSE;
	mxStopDirect:=FALSE;
	mxStopcycleEmpty:=False;
	
	HydraulicPump.M_Stop();
	CoolingFan.M_Stop();
	FilterMotor.M_Stop();
	AccuDrainValve.M_Off();
	IsolationValve.M_Off();
	PressurizePumpValve.M_Off();
END_IF

mxCycleHasError:=FALSE;

T_DelayOpenBlockingValve(PT:= T#15S);
T_DepresurizePump(PT:=T#2S);

mxHydraulicsReady:= miCycleState=8;


(*Cycle State's*)
CASE miCycleState OF

	0:	// Idle state/Wait for start
		IF mxStopDirect THEN
			mxStopDirect:= FALSE;		
			miCycleState:= 15;
		ELSIF mxStopCycle THEN		
			miCycleState:= 0;
			mxStopCycle:=FALSE;
		ELSIF mxStartCycle THEN		
			miCycleState:= 1;
			mxStartCycle:=FALSE;
			mxStopCycleEmpty:=FALSE;
		END_IF	

	1:	// Check oil temperature and oil levels	and valves Start main pump
		IF mxStopDirect THEN
			mxStopDirect:= FALSE;
			miCycleState:= 15;
		ELSIF mxStopCycle THEN
			mxStopCycle:= FALSE;
			miStopState:= miCycleState;
			miCycleState:= 13;
		ELSIF ixTemperatureSwitchTooHigh AND ixOilLvlTooLow AND NOT PressurizePumpValve.mxIsOn THEN			
			HydraulicPump.M_Start();
			miCycleState:= 2;
		END_IF

	2:	//When pump is running, start cooler and filterpump 	
		IF mxStopDirect THEN
			mxStopDirect:= FALSE;
			miCycleState:= 15;
		ELSIF mxStopCycle THEN
			mxStopCycle:= FALSE;
			miStopState:= miCycleState;
			miCycleState:= 13;
		ELSIF HydraulicPump.IsRunning THEN			
			FilterMotor.M_Start();
			miCycleState:= 3;
		END_IF

	3:	//When pumps are running open the Pressurize valve 
		IF mxStopDirect THEN
			mxStopDirect:= FALSE;			
			miCycleState:= 15;
		ELSIF mxStopCycle THEN
			mxStopCycle:= FALSE;
			miStopState:= miCycleState;
			miCycleState:= 13;
		ELSIF FilterMotor.IsRunning THEN					
			PressurizePumpValve.M_On();
			miCycleState:= 4;
		END_IF
	
	4:	// When circulation valve is open, open accumulator valve
		IF mxStopDirect THEN
			mxStopDirect:= FALSE;		
			miCycleState:= 15;
		ELSIF mxStopCycle THEN
			mxStopCycle:= FALSE;
			miStopState:= miCycleState;
			miCycleState:= 13;
		ELSIF PressurizePumpValve.mxIsOn THEN			
			AccuDrainValve.M_On();
			miCycleState:= 5;
		END_IF
	
	5:	//Check if accuValve is open and wait for 15s 
		IF mxStopDirect THEN
			mxStopDirect:= FALSE;		
			miCycleState:= 15;
		ELSIF mxStopCycle THEN
			mxStopCycle:= FALSE;
			miStopState:= miCycleState;
			miCycleState:= 13;
		ELSIF AccuDrainValve.mxIsOn THEN			
			T_DelayOpenBlockingValve.IN:=TRUE;
			miCycleState:= 6;
		END_IF
		
	6:	//Open blocking valve
		IF mxStopDirect THEN
			mxStopDirect:= FALSE;	
			miCycleState:= 15;
		ELSIF mxStopCycle THEN
			mxStopCycle:= FALSE;
			miStopState:= miCycleState;
			miCycleState:= 13;
		ELSIF T_DelayOpenBlockingValve.Q THEN				
			T_DelayOpenBlockingValve.IN:=FALSE;
			IsolationValve.M_On();
			miCycleState:= 7;
		END_IF
		
	7:	// Check if blocking valve is open and main pressure is > X 
		IF mxStopDirect THEN
			mxStopDirect:= FALSE;
			miCycleState:= 15;
		ELSIF mxStopCycle THEN
			mxStopCycle:= FALSE;
			miStopState:= miCycleState;
			miCycleState:= 13;
		ELSIF IsolationValve.mxIsOn AND (MainSystemPressure.EngFilt > 240.0) THEN			
			miCycleState:= 8;
		END_IF
		
	8: // State of main hydraulics is running, wait in this step for stop.	
		IF mxStopDirect THEN
			mxStopDirect:= FALSE;
			miCycleState:= 15;
		ELSIF mxStopCycle THEN		
			mxStopCycle:= FALSE;
			miStopState:= miCycleState;
			miCycleState:= 13;
		
		// Stopping the cycle CMD.
		ELSIF mxStopCycleEmpty THEN
			mxStopCycleEmpty:=FALSE;
			miStopState:= miCycleState;
			miCycleState:= 9;
		END_IF
		
	9:	// Check if all analog valves are in safe state. (not controlled)
		IF mxStopDirect THEN
			mxStopDirect:= FALSE;
			miCycleState:= 15;
		ELSIF mxStopCycle THEN		
			mxStopCycle:= FALSE;
			miStopState:= miCycleState;
			miCycleState:= 13;
		ELSIF (MAIN.InMoldDrying.TopMoldA.HydraulicCilinder.SafePosReached AND 
			Main.InMoldDrying.TopMoldB.HydraulicCilinder.SafePosReached AND 
			Main.InMoldDrying.TransferMold.HydraulicCilinder.SafePosReached) THEN
			PressurizePumpValve.M_Off();	// Pomp vrijschakelen
			CoolingFan.M_Stop();
			FilterMotor.M_Stop();
			
			T_DepresurizePump.IN := TRUE;
			
			miCycleState:=10;
		END_IF
		
	10:	// Check if pressurise pump valve, coolingfan / filtermotor are stopped/closed -> Open isolation and drain valve
		IF mxStopDirect THEN
			mxStopDirect:= FALSE;
			miCycleState:= 15;
		ELSIF mxStopCycle THEN		
			mxStopCycle:= FALSE;
			miStopState:= miCycleState;
			miCycleState:= 13;
		ELSIF NOT PressurizePumpValve.mxIsOn AND NOT CoolingFan.IsRunning AND NOT FilterMotor.IsRunning AND T_DepresurizePump.Q THEN
			T_DepresurizePump.IN := FALSE;	
			IsolationValve.M_Off();
			AccuDrainValve.M_Off();
			micycleState:=11;
		END_IF
		
	11:	// Check if isolationvalve and accudrain valve have stopped -> stop pump
		IF mxStopDirect THEN
			mxStopDirect:= FALSE;
			miCycleState:= 15;
		ELSIF mxStopCycle THEN		
			mxStopCycle:= FALSE;
			miStopState:= miCycleState;
			miCycleState:= 13;
		ELSIF NOT IsolationValve.mxIsOn AND NOT AccuDrainValve.mxIsOn THEN	
			HydraulicPump.M_Stop();
			miCycleState:=0;
		END_IF
		
	13:	// Stop cycle, wait for start 
		IF mxStopDirect THEN
			mxStopDirect:= FALSE;
			miCycleState:= 15;
		ELSE
 			IsolationValve.M_Off();		// Switch off the isolation valve in rest mode (rest of hydraulics keep functioning as normal).
			miCycleState:=14;
		END_IF
		
	14: // Pause cycle step.			// in rest.
		IF mxStopDirect OR MAIN.Errors.InMoldDryingErrors.TopMoldA.Hydraulic.SafePositionValveNotReached OR
		Main.Errors.InMoldDryingErrors.TopMoldB.Hydraulic.SafePositionValveNotReached OR
		Main.Errors.InMoldDryingErrors.TransferMold.HydraulicCilinder.SafePositionValveNotReached THEN
			mxStopDirect:= FALSE;
			miCycleState:= 15;
		ELSIF mxStartCycle THEN
			mxStopCycle:=FALSE;
			mxStartCycle:=FALSE;
 			IsolationValve.M_on();		// At restart, open valve again.
			miCycleState:=miStopState;
		ELSIF mxStopCycleEmpty THEN		// At pause stop rest of hydraulics.
			mxStopcycleEmpty:=FALSE;
			miCycleState := 9;
		END_IF

	15:	// Stop Direct
		mxStartCycle:= FALSE;
		mxStopCycle:= FALSE;
		mxStopCycleEmpty:=FALSE;
		mxInitialized:= FALSE;
		
		HydraulicPump.M_Stop();
		CoolingFan.M_Stop();
		FilterMotor.M_Stop();
		
		IsolationValve.M_Off();
		PressurizePumpValve.M_Off();
		AccuDrainValve.M_Off();		
		
		miCycleState:= 0;
END_CASE

mxCycleBusy:= miCycleState<>0;
mxCycleInPause := miCycleState=14;
END_ACTION

ACTION Error:

SR_TempTooHigh(SET1:=NOT ixTemperatureSwitchTooHigh, RESET:=mxReset , Q1=>Errors.OilTemperatureTooHigh);
SR_LevelTooLow(SET1:=NOT ixOilLvlTooLow, Reset:=mxReset, Q1=>Errors.OilLevelTooLow);

SR_Filter100Dirty(SET1:=NOT ixPressureFilterAt100, RESET:=mxReset, Q1=>Errors.Filter100Dirty);
SR_AuxFilter100Dirty(SET1:=NOT ixAuxFilterAt100, RESET:=mxReset, Q1=>Errors.AuxFilter100Dirty);

SR_Filter75DirtyWarning(SET1:=ixPressureFilterAt75, RESET:=mxReset, Q1=>Errors.Filter75Dirty);
SR_AuxFilter75DirtyWarning(SET1:=ixAuxFilterAt75, RESET:=mxReset, Q1=>Errors.AuxFilter75Dirty);

SR_CabinetCoolerError(SET1:= NOT ixCabinetCoolerError, Reset:=mxReset, Q1=>);

SR_HydraulicsMcc24VError(SET1:= NOT ixHydraulicsMcc24vError, Reset:=mxReset, Q1=>);


RT_Doorsopenend(CLK:=mxDoorOpened);
RT_EmergencyStop(CLK:=mxEmergency);

IF RT_Doorsopenend.Q THEN
	M_StopCycle();
END_IF

IF RT_EmergencyStop.Q THEN
	M_StopDirect();
END_IF



(**********************************************************************************************************)
mxErrorStopinPos:= HydraulicPump.mxErrorStopinPos OR FilterMotor.mxErrorStopinPos OR CoolingFan.mxErrorStopinPos;

mxErrorInit:= HydraulicPump.mxErrorInit OR Errors.Filter100Dirty OR Errors.AuxFilter100Dirty OR Errors.OilLevelTooLow OR
				Errors.OilTemperatureTooHigh OR FilterMotor.mxErrorInit OR CoolingFan.mxErrorInit;
END_ACTION

METHOD M_StartCycle : BOOL
IF NOT mxCycleBusy OR mxCycleInPause THEN
	mxStartCycle:= TRUE;	
	mxStopCycle:=False;
END_IF
END_METHOD

METHOD M_StopCycle : BOOL
IF mxCycleBusy THEN 
	mxStopCycle:= TRUE; 
END_IF
END_METHOD

METHOD M_StopCycleEmpty : BOOL
IF mxCycleBusy THEN 
	mxStopCycleEmpty:= TRUE; 
END_IF
END_METHOD

METHOD M_StopDirect

IF mxCycleBusy THEN
	mxStopDirect:= TRUE;	
END_IF
END_METHOD

METHOD M_StopInit
;
END_METHOD

ACTION Objects:
OilTemperature(
	EngLowLimit:= -25, 
	EngUpperLimit:= 100); (* In °C *)

PressurizePumpValve(
	mxReset:= mxReset, 
	mxEmergency:=mxEmergency , 
	mxAutoMode:=mxAutoMode , 
	RHSR_Blocked:= , 
	SlowValveIsInverted:= , 
	mxDisableManualAutoTrigger:=TRUE,
	mxIsOn=> );
	
	
	// special situation, on door opened keep the accu drain valve openend.
AccuDrainValve(
	mxReset:= mxReset, 
	mxEmergency:= mxDoorOpened, 
	mxAutoMode:=mxAutoMode , 
	RHSR_Blocked:= , 
	SlowValveIsInverted:= , 
	mxDisableManualAutoTrigger:=TRUE,
	mxIsOn=> );
	
IsolationValve(
	mxReset:= mxReset, 
	mxEmergency:=mxEmergency , 
	mxAutoMode:=mxAutoMode , 
	RHSR_Blocked:= , 
	SlowValveIsInverted:= , 
	mxDisableManualAutoTrigger:=TRUE,
	mxIsOn=> );
	
HydraulicPump(
	mxReset:= mxReset, 
	mxEmergency:= mxEmergency,
	mxAutoMode:= mxAutoMode,
	mxDisableManualAutoTrigger:=TRUE,
	Errors=> Errors.HydraulicPump);
	
FilterMotor(
	mxReset:= mxReset, 
	mxEmergency:= mxEmergency, 
	mxAutoMode:= mxAutoMode, 
	mxDisableManualAutoTrigger:=TRUE,
	Errors=>Errors.FilterMotor);
	
CoolingFan(
	mxReset:= mxReset, 
	mxEmergency:= mxEmergency,
	mxAutoMode:= mxAutoMode,
	mxDisableManualAutoTrigger:=TRUE,
	Errors=> Errors.Coolingfan);
	
MainSystemPressure(
	EngLowLimit:=0, 
	EngUpperLimit:=315, 
	maOut=> , 
	EngUnits=> , 
	EngFilt=> , 
	OverRange=> , 
	UnderRange=> );
END_ACTION

END_FUNCTION_BLOCK

// ---- POUs/Standard/Motor/FB_MotorSS.TcPOU
FUNCTION_BLOCK FB_MotorSS
VAR_INPUT
	mxReset							: BOOL;
	mxEmergency						: BOOL;
	mxAutoMode						: BOOL;
	mxDisableManualAutoTrigger		: BOOL := FALSE; // If this bit is enabled, the outputs status is not changed when change from/to automode happens
END_VAR
VAR_OUTPUT
(*Errors*)
	Errors							: ST_MotorSSErrors;
	mxErrorInit						: BOOL;		(* Error, stop immediately. Initialisation neccesary *)
	mxErrorStopinPos				: BOOL;		(* Error, stop in position. Only reset neccesary *)

(* State vars *)
	mxCycleBusy						: BOOL;
	mxInitBusy						: BOOL;
	
(* Vars *)
	mxInitialized					: BOOL;
	IsRunning						: BOOL;
	
END_VAR
VAR
	ixSSFailure						AT %I* : BOOL;
	ixMaintenance					AT %I* : BOOL;
	ixIsRunning						AT %I* : BOOL;
	Q								AT %Q* : BOOL;
	
	Hmi_On							: BOOL;
	RT_AutoMode						: R_TRIG;
	SR_ErrorMaintenance				: SR;
	SR_ErrorSS: SR;
	mxTest: BOOL;
END_VAR

Error();

(* Reset hmi when switched to automode*)
RT_AutoMode(CLK:= mxAutoMode);

// if manual mode becomes active, the manualmode (hmi) is over written by its current state.
// this ensures that the motor keeps running when it was running and is switched to manual. 
IF RT_AutoMode.Q AND NOT mxDisableManualAutoTrigger THEN Hmi_On:= Q; END_IF	

(* Manual control *)
//IF NOT mxAutoMode THEN Q:= Hmi_On; END_IF

IsRunning:= ixIsRunning;

ACTION Error:
SR_ErrorSS(SET1:= NOT ixSSFailure, RESET:= mxReset, Q1=> Errors.SofstarterFailure);
SR_ErrorMaintenance(SET1:= NOT ixMaintenance, RESET:= mxReset, Q1=> Errors.Maintenance);

(******************************************************************************************************)
mxErrorStopinPos:= FALSE;
mxErrorInit:= Errors.SofstarterFailure OR Errors.Maintenance;
END_ACTION

METHOD M_Init

Q:= FALSE;
END_METHOD

METHOD M_Start : BOOL
VAR_INPUT
END_VAR
Q:=TRUE;

(* Return Value *)
M_Start:= Q;
END_METHOD

METHOD M_Stop : BOOL
VAR_INPUT
END_VAR
Q:= FALSE;

(* Return Value *)
M_Stop:= NOT Q;
END_METHOD

END_FUNCTION_BLOCK

// ---- POUs/Standard/Motor/FB_Motor.TcPOU
FUNCTION_BLOCK FB_Motor
VAR_INPUT
	mxReset							: BOOL;
	mxEmergency						: BOOL;
	mxAutoMode						: BOOL;
	mxDisableManualAutoTrigger		: BOOL := FALSE; // If this bit is enabled, the outputs status is not changed when change from/to automode happens
END_VAR
VAR_OUTPUT
(*Errors*)
	Errors							: ST_MotorErrors;
	mxErrorInit						: BOOL;		(* Error, stop immediately. Initialisation neccesary *)
	mxErrorStopinPos				: BOOL;		(* Error, stop in position. Only reset neccesary *)

(* State vars *)
	mxCycleBusy						: BOOL;
	mxInitBusy						: BOOL;
	
(* Vars *)
	mxInitialized					: BOOL;
	IsRunning						: BOOL;
	
END_VAR
VAR
	ixThermal						AT %I* : BOOL;
	ixRunning						AT %I* : BOOL;
	ixMaintenance					AT %I* : BOOL;
	Q								AT %Q* : BOOL;
	
	Hmi_On							: BOOL;
	RT_AutoMode						: R_TRIG;
	SR_ErrorThermal					: SR;
	SR_ErrorMaintenance				: SR;
	Ixtest: BOOL;
END_VAR

Error();

(* Reset hmi when switched to automode*)
RT_AutoMode(CLK:= mxAutoMode);

// if manual mode becomes active, the manualmode (hmi) is over written by its current state.
// this ensures that the motor keeps running when it was running and is switched to manual. 
IF RT_AutoMode.Q AND NOT mxDisableManualAutoTrigger THEN Hmi_On:= Q; END_IF	

(* Manual control *)
//IF NOT mxAutoMode THEN Q:= Hmi_On; END_IF

// Is running becomes high when signal becomes low.
IsRunning:= NOT ixRunning;

ACTION Error:
SR_ErrorThermal(SET1:= NOT ixThermal, RESET:= mxReset, Q1=> Errors.Thermal);
SR_ErrorMaintenance(SET1:= NOT ixMaintenance, RESET:= mxReset, Q1=> Errors.Maintenance);

(******************************************************************************************************)
mxErrorStopinPos:= FALSE;
mxErrorInit:= Errors.Thermal OR Errors.Maintenance;
END_ACTION

METHOD M_Init

Q:= FALSE;
END_METHOD

METHOD M_Start : BOOL
VAR_INPUT
END_VAR
Q:=TRUE;

(* Return Value *)
M_Start:= Q;
END_METHOD

METHOD M_Stop : BOOL
VAR_INPUT
END_VAR
Q:= FALSE;

(* Return Value *)
M_Stop:= NOT Q;
END_METHOD

END_FUNCTION_BLOCK

// ---- POUs/ProductHandling/FB_ProductHandling.TcPOU
FUNCTION_BLOCK FB_ProductHandling
VAR CONSTANT
	sCycleStateTextDef: ARRAY[0..30]  OF STRING :=	
		['State 0: Wait for Start',
		'State 1: Gantry A, Gantry B and Product conveyor started',
		'State 2: ',
		'3',
		'4',
		'5',
		'6',
		'7',
		'8',
		'9',
		'State 10:',
		'State 11:',
		'State 12:',
		'State 13:',
		'State 14:',
		'State 15:',
		'State 16:',
		'State 17:',
		'State 18:',
		'State 19:',
		'State 20: Stopcylce waiting for EAMC ready',
		'State 21: Stop cycle awaiting gantries ready',
		'State 22: Stop cycle awaiting outfeed conveyor ready',
		'State 23: Stop cycle Stopping Gantries and conveyor',
		'State 24: Stop cycle awaiting restart',
		'State 25: Stop direct'];
	
	tCycleStateTimeouts: ARRAY[0..10] OF TIME := 
		[T#10S,T#10S,T#10S,T#10S,T#10S,T#10S,T#10S,T#10S,T#10S,T#10S,
		T#10S];

	sInitStateTextDef: ARRAY[0..10] OF STRING :=
		['State 0: Wait for Start',
		'State 1: Description Init State 1',
		'State 2: Description Init State 2',
		'State 3; Description Init State 3',
		'State 4; Description Init State 4',
		'State 5; Description Init State 5',
		'State 6; Error State'];

	tInitStateTimeouts: ARRAY[0..10] OF TIME := 
		[T#10S,T#10S,T#10S,T#10S,T#10S,T#10S,T#10S,T#10S,T#10S,T#10S
		,T#10S];
END_VAR
VAR_INPUT
	mxResetCycleState				: BOOL;
	mxResetInitState				: BOOL;
	mxForceInit						: BOOL; (*Reset Calibration Flag*)
	mxReset							: BOOL;	(*Reset Error*)
	mxEmergency						: ARRAY [1..Max_Zones+1] OF BOOL; // 1=TakeOutA, 2=Aside, 3=mid, 4=Bside, 5=TakeoutB, 6= GantryB, 7=GantryA, 8=All EM stop.
	mxAutoMode						: BOOL; (* TRUE = Automode *)
	mxFirstCycle					: BOOL;
	mxSideA_Enabled					: BOOL;
	mxSideB_Enabled					: BOOL;
	mxEamcIsEmpty					: BOOL;
	mxProductReadyAtTakeout_A		: BOOL;
	mxProductReadyAtTakeout_B		: BOOL;
	
	mxPause							: BOOL;
END_VAR
VAR_IN_OUT
	MachParameters					: ST_ProductHandlingMachPar;
	ProdParameters					: ST_ProductHandlingProdPar;
	SysParameters					: ST_ProductHandlingSysPar;
END_VAR
VAR_OUTPUT
(*Errors*)
	Errors							: ST_ProductHandlingErrors;
	mxErrorInit						: BOOL;		(* Error, stop immediately. Initialisation neccesary *)
	mxErrorStopinPos				: BOOL;		(* Error, stop in position. Only reset neccesary *)

(* State vars *)
	mxCycleBusy						: BOOL;
	mxInitBusy						: BOOL;
	
(* Vars *)
	mxInitialized					: BOOL;
	mxProductPickedUpGantry_A		: BOOL;
	mxProductPickedUpGantry_B		: BOOL;
	mxGantrysNotBusy				: BOOL;
	
END_VAR
VAR
	(* State vars *)
	miCycleState					: INT :=0;
	miCycleOldstate					: INT :=0;
	mxCycleTransitionState			: BOOL := FALSE;
	sCycleStateText					: STRING;
	exCycleTimeOut					: BOOL;		(* Timeout for the whole programcycle *)
	CycleTimeout					: TON;
	CycleTimeOutUpFlank				: R_TRIG;
	mxCycleTimeoutEnable			: BOOL;
	CycleTime						: REAL;
	mxCycleHasError					: BOOL;
	miStopState						: INT;
	mxStartCycle					: BOOL;
	mxStopCycle						: BOOL;
	mxStopDirect					: BOOL;
	
	miInitState						: INT	:=0;
	miInitOldstate					: INT	:=0;
	mxInitTransitionState			: BOOL	:= FALSE;
	sInitStateText					: STRING;
	exInitTimeOut					: BOOL;		(* Timeout for the whole programcycle *)
	InitTimeout						: TON;
	InitTimeOutUpFlank				: R_TRIG;
	mxInitTimeoutEnable				: BOOL;
	InitTime						: REAL;
	mxInitHasError					: BOOL;
	mxStartInit						: BOOL;
	mxStopInit						: BOOL;

	(*Errors *)
	SR_HorMovingVertNotAtTranspPos_A	: SR;(* RedHot SafetyRule, Horizontal is moving when vertical is not at transport position *)
	SR_HorMovingVertNotAtTranspPos_B	: SR;(* RedHot SafetyRule, Horizontal is moving when vertical is not at transport position *)
	SR_VertMovingHorNotInPos_A			: SR;(* RedHot SafetyRule, Vertical is moving when horizontal is not at pick or drop position *)
	SR_VertMovingHorNotInPos_B			: SR;(* RedHot SafetyRule, Vertical is moving when horizontal is not at pick or drop position *)

	(* Objects *)
	GantryA								: FB_Gantry;
	GantryB								: FB_Gantry;
	OutfeedConveyor						: FB_OutfeedConveyor;
	
	mxHMI_DisableCollision				: BOOL;

	RT_ProductReadyAtTakeout_A: R_TRIG;
	RT_ProductReadyAtTakeout_B: R_TRIG;
	mxHorOnPos_A: BOOL;
	mxHorOnPos_B: BOOL;
	
	RT_AutoMode: R_TRIG;
	mxSafetyRulesEnabled: BOOL;
	T_StopCommisioningMode: TON;
	mxVertOnPos_A: BOOL;
	mxVertOnPos_B: BOOL;
	mxStopCycleEmpty: BOOL;
	
	
	mxInPause : BOOL;
END_VAR

(* Stopcycle = empty machine *)
(* Pause = stop at place *)

Error();
Cycle();
Init();
Objects();

RT_AutoMode(CLK:= mxAutoMode);
IF RT_AutoMode.Q THEN
	mxHMI_DisableCollision:= FALSE;
END_IF

T_StopCommisioningMode(IN:=MachParameters.CommisioningMode, PT:=T#120M);
IF T_StopCommisioningMode.Q THEN
	MachParameters.CommisioningMode := FALSE;
END_IF

ACTION Cycle:
(*StateChange (Transition)  Signalgeneration*)
mxCycleTransitionState:=(miCycleState<>miCycleOldstate);
(*State text*)
sCycleStateText:=sCycleStateTextDef[miCycleState];
(*Timeout Watchdog for Statemachine*)
mxCycleTimeoutEnable:=NOT (miCycleState=0) AND NOT mxReset;

CycleTimeout(IN:=mxCycleTimeoutEnable, PT:=tCycleStateTimeouts[miCycleState] );
CycleTimeOutUpFlank(CLK:=CycleTimeout.Q );
miCycleOldstate:=miCycleState;

(*Set Errorbit when Raising edge of Timeout has been detected*)
IF CycleTimeOutUpFlank.Q THEN
	exCycleTimeOut:=TRUE; 			(* 1 Timeout for the whole programcycle *)
END_IF

(*Function to reset the Statemachine*)
IF mxResetCycleState THEN
	mxResetCycleState:= FALSE;
	miCycleState:=0;
	miCycleOldstate:=miCycleState;
	mxCycleTransitionState:=FALSE;

	mxInitialized:= FALSE;
	mxStartCycle:= FALSE;
	mxStopCycle:= FALSE;
	mxStopCycleEmpty := FALSE;
	mxStopDirect:= FALSE;

	mxEamcIsEmpty:= FALSE;
	mxPause:= FALSE;
			
	GantryA.mxResetCycleState:= TRUE;
	GantryB.mxResetCycleState:= TRUE;
	OutfeedConveyor.mxResetCycleState:= TRUE;

END_IF

(*Definition State has Error*)
mxCycleHasError:=FALSE;

RT_ProductReadyAtTakeout_A(CLK:= mxProductReadyAtTakeout_A);
RT_ProductReadyAtTakeout_B(CLK:= mxProductReadyAtTakeout_B);

(*Cycle State's*)
CASE miCycleState OF
	0:
	(*
		- Wait for startcycle
		- Start GantryA, B, Outfeedconveyor

	Als Stop dan leegdraaien, dus wachten op EAMC die leeg is
	Als Pause dan alles stopInPos en vrijgeven. 
		*  
	*)
		IF mxStartCycle THEN
			mxStartCycle:= FALSE;

			IF mxSideA_Enabled THEN GantryA.M_StartCycle(); END_IF
			IF mxSideB_Enabled THEN GantryB.M_StartCycle(); END_IF
			OutfeedConveyor.M_StartCycle();
			
			miCycleState:= 1;
		END_IF	

	(* Gantry A, Gantry B, Outfeed started *)
	1:
		IF RT_ProductReadyAtTakeout_A.Q THEN
			GantryA.mxProductReadyAtTakeout:= TRUE;
		END_IF
		IF RT_ProductReadyAtTakeout_B.Q THEN
			GantryB.mxProductReadyAtTakeout:= TRUE;
		END_IF
	
		IF mxStopCycleEmpty AND mxEamcIsEmpty THEN (* Emtpy *)
			mxStopCycleEmpty:= FALSE;
			
			miStopState:= miCycleState;
			miCycleState:= 20;
		ELSIF mxStopCycle THEN
			mxStopCycle:= FALSE;			

			(* Stop Cycle *)
			IF mxSideA_Enabled THEN GantryA.M_StopCycle(); END_IF
			IF mxSideB_Enabled THEN GantryB.M_StopCycle(); END_IF
			OutfeedConveyor.M_StopCycle();
			
			miStopState:= miCycleState;
			miCycleState:= 23;
		END_IF

	(* Stop Cycle, wait for EAMC is empty *)
	20:
		IF mxStopDirect THEN
			mxStopDirect:= FALSE;
			
			miCycleState:= 25;
		ELSIF mxEamcIsEmpty THEN // Signal from EAMC that the machine is empty, Gantry A B signals are set when product ready at gantry
		
			miCycleState:= 21;			
		END_IF

	(* Stop Cycle, wait for Gantry is empty *)
	21:
		IF mxStopDirect THEN
			mxStopDirect:= FALSE;
			
			miCycleState:= 25;
		ELSIF (GantryA.mxIsEmpty OR NOT mxSideA_Enabled) AND (GantryB.mxIsEmpty OR NOT mxSideB_Enabled) THEN
		
			(* Stop Cycle *)
			IF mxSideA_Enabled THEN GantryA.M_StopCycle(); END_IF
			IF mxSideB_Enabled THEN GantryB.M_StopCycle(); END_IF
			OutfeedConveyor.M_StopCycle();
			
			miCycleState:= 22;
		END_IF

	(* Stop Cycle, outfeed conveyor empty *)
	22:
		IF mxStopDirect THEN
			mxStopDirect:= FALSE;
			
			miCycleState:= 25;
		ELSIF NOT OutfeedConveyor.mxCycleBusy THEN
		
			miCycleState:= 0;
		END_IF
	
	(* Stop Cycle, Stop gantry's, Belt *)
	23:
		IF mxStopDirect THEN
			mxStopDirect:= FALSE;
			
			miCycleState:= 25;
		ELSIF NOT GantryA.mxCycleBusy AND NOT GantryB.mxCycleBusy AND NOT OutfeedConveyor.mxCycleBusy THEN
			
			miCycleState:= 24;
		END_IF

	(* Stop Cycle, wait for restart *)
	24:
		IF mxStopDirect THEN
			mxStopDirect:= FALSE;
			
			miCycleState:= 25;
		ELSIF mxStartCycle THEN
			mxStartCycle:= FALSE;
			
			miCycleState:= miStopState;
		END_IF

	(* Stop Direct *)
	25:
		mxInitialized:= FALSE;
		mxStartCycle:= FALSE;
		mxStopCycle:= FALSE;
		mxStopDirect:= FALSE;

		GantryA.M_StopDirect();
		GantryB.M_StopDirect();
		OutfeedConveyor.M_StopDirect();
		
		miCycleState:= 0;
END_CASE

mxCycleBusy:= miCycleState<>0 AND NOT (miCycleState=22);
END_ACTION

ACTION Error:
(* Red Hot Safety *)

mxSafetyRulesEnabled := (mxInitialized AND mxAutoMode) OR (NOT mxAutomode); //AND NOT MachParameters.CommisioningMode;

mxHorOnPos_A:= (GantryA.mrActPosHorizontal <= (MachParameters.GantryA.PositionHorizontalPickup + 10) AND GantryA.mrActPosHorizontal >= (MachParameters.GantryA.PositionHorizontalPickup - 10)) OR
	 	(GantryA.mrActPosHorizontal <= (MachParameters.GantryA.PositionHorizontalDropOff + 10) AND GantryA.mrActPosHorizontal >= (MachParameters.GantryA.PositionHorizontalDropOff - 10));

mxHorOnPos_B:=(GantryB.mrActPosHorizontal <= (MachParameters.GantryB.PositionHorizontalPickup + 10) AND GantryB.mrActPosHorizontal >= (MachParameters.GantryB.PositionHorizontalPickup - 10)) OR
	 	(GantryB.mrActPosHorizontal <= (MachParameters.GantryB.PositionHorizontalDropOff + 10) AND GantryB.mrActPosHorizontal >= (MachParameters.GantryB.PositionHorizontalDropOff - 10));

mxVertOnPos_A := (GantryA.mrActPosVertical <= (MachParameters.GantryA.Vert_PositionTransport - 10) AND GantryA.mrActPosVertical >= (MachParameters.GantryA.Vert_PositionTransport + 5));

mxVertOnPos_B := (GantryB.mrActPosVertical <= (MachParameters.GantryB.Vert_PositionTransport - 10) AND GantryB.mrActPosVertical >= (MachParameters.GantryB.Vert_PositionTransport + 5));
		


SR_HorMovingVertNotAtTranspPos_A(
	SET1:= mxSafetyRulesEnabled AND mxAutoMode AND GantryA.mxHorizontalIsMoving AND mxVertOnPos_A, 
	RESET:= mxReset, Q1=> Errors.RH_HorMovingVertNotAtTranspPos_A);
	
SR_HorMovingVertNotAtTranspPos_B(
	SET1:=mxSafetyRulesEnabled AND mxAutoMode AND GantryB.mxHorizontalIsMoving AND mxVertOnPos_B,
	RESET:= mxReset, Q1=> Errors.RH_HorMovingVertNotAtTranspPos_B);

SR_VertMovingHorNotInPos_A(
	SET1:=mxSafetyRulesEnabled AND mxAutoMode AND GantryA.mxVerticalIsMoving AND NOT mxHorOnPos_A, 
	RESET:= mxReset, Q1=> Errors.RH_VertMovingHorNotInPos_A);

SR_VertMovingHorNotInPos_B(
	SET1:=mxSafetyRulesEnabled AND mxAutoMode AND GantryB.mxVerticalIsMoving AND NOT mxHorOnPos_B, 
	RESET:= mxReset, Q1=> Errors.RH_VertMovingHorNotInPos_B);

(*************************************************************************************************)
mxErrorInit:= GantryA.mxErrorInit OR GantryB.mxErrorInit OR OutfeedConveyor.mxErrorInit OR 
				Errors.RH_HorMovingVertNotAtTranspPos_A OR Errors.RH_HorMovingVertNotAtTranspPos_B OR 
				Errors.RH_VertMovingHorNotInPos_A OR Errors.RH_VertMovingHorNotInPos_B;
				
mxErrorStopinPos:= GantryA.mxErrorStopinPos OR GantryB.mxErrorStopinPos OR OutfeedConveyor.mxErrorStopinPos;
END_ACTION

ACTION Init:
(*StateChange (Transition)  Signalgeneration*)
mxInitTransitionState:=(miInitState<>miInitOldstate);
(*State text*)
sInitStateText:=sInitStateTextDef[miInitState];
(*Timeout Watchdog for Statemachine*)
mxInitTimeoutEnable:=NOT (miInitState=0)  AND NOT mxReset;

InitTimeout(IN:=mxInitTimeoutEnable  , PT:=tInitStateTimeouts[miInitState] );
InitTimeOutUpFlank(CLK:=InitTimeout.Q );
miInitOldstate:=miInitState;

(*Set Errorbit when Raising edge of Timeout has been detected*)
IF InitTimeOutUpFlank.Q THEN
	exInitTimeOut:=TRUE; 			(* 1 Timeout for the whole programcycle *)
END_IF

(*Function to reset the Statemachine*)
IF mxResetInitState THEN
	mxResetInitState:=FALSE;
	miInitState:=0;
	miInitOldstate:=miInitState;
	mxInitTransitionState:=FALSE;

	mxInitialized:= FALSE;
	mxStartInit:= FALSE;
	mxStopInit:= FALSE;
	
	GantryA.mxResetInitState:= TRUE;
	GantryA.mxResetCycleState:=TRUE;
	GantryB.mxResetInitState:=TRUE;
	GantryB.mxResetCycleState:= TRUE;
	OutFeedConveyor.mxResetInitState:=TRUE;
	OutfeedConveyor.mxResetCycleState:= TRUE;	
END_IF

(*Definition State has Error*)
mxInitHasError:=FALSE;

(*Init State's*)
CASE miInitState OF
	0:
	
	(* 
		- Wait for start int
		- Blow off uit
		- vacuum aan laten
		- Vertical move up to transport pos.
		- Horizontal move back to drop off positie
		- 	
	
	*)
		IF mxStartInit THEN
			mxStartInit:= FALSE;
			mxInitialized:= FALSE;
		
			miInitState:= 1;
		END_IF

	1:
		IF mxStopInit THEN
			mxStopInit:= FALSE;
			miInitState:= 10;
		ELSE
			IF mxSideA_Enabled THEN GantryA.M_StartInit(); END_IF			
			IF mxSideB_Enabled THEN GantryB.M_StartInit(); END_IF
			OutfeedConveyor.M_StartInit();

			miInitState:= 2;
		END_IF

	2:
		IF mxStopInit THEN
			mxStopInit:= FALSE;
			miInitState:= 10;
		ELSIF (GantryA.mxInitialized OR NOT mxSideA_Enabled) AND (GantryB.mxInitialized OR NOT mxSideB_Enabled)
				 AND OutfeedConveyor.mxInitialized THEN
	
			mxInitialized:= TRUE;
			miInitState:= 0;
		END_IF

	(* Stop Init *)
	10:
		mxStartInit:= FALSE;
		mxStopInit:= FALSE;
		mxInitialized:= FALSE;

		GantryA.M_StopInit();
		GantryB.M_StopInit();
		OutfeedConveyor.M_StopInit();
		
		miInitState:= 0;
			
END_CASE

mxInitBusy:= miInitState<>0;
END_ACTION

METHOD M_StartCycle

IF (NOT mxCycleBusy AND mxInitialized) OR (mxInPause AND mxInitialized) THEN
	mxInPause:=FALSE;
	mxStartCycle:= TRUE;	
END_IF
END_METHOD

METHOD M_StartInit

IF NOT mxInitBusy THEN 
	mxStartInit:= TRUE; 
END_IF
END_METHOD

METHOD M_StopCycle

IF mxCycleBusy THEN
	mxStopCycle:= TRUE;	
	mxInPause:=TRUE;
END_IF
END_METHOD

METHOD M_StopCycleEmpty

IF mxCycleBusy THEN 
	mxStopCycleEmpty:= TRUE; 
END_IF
END_METHOD

METHOD M_StopDirect

IF mxCycleBusy THEN
	mxStopDirect:= TRUE;	
END_IF
END_METHOD

METHOD M_StopInit

IF mxInitBusy THEN 
	mxStopInit:= TRUE; 
END_IF
END_METHOD

ACTION Objects:
GantryA(
	mxReset:= mxReset, 
	mxEmergency:= mxEmergency[1] OR mxEmergency[2] OR mxEmergency[7], 
	mxAutoMode:= mxAutoMode, 
	mxFirstCycle:= mxFirstCycle,
	mrModPosConveyor:= OutfeedConveyor.mrActModPos, 
	mxDisableCollision:= mxHMI_DisableCollision,
	MachParameters:= MachParameters.GantryA, 
	ProdParameters:= ProdParameters.GantryA, 
	SysParameters:= SysParameters.GantryA,
	mxProductPickedUp=> mxProductPickedUpGantry_A,
	Errors=> Errors.Gantry_A);
	
GantryB(
	mxReset:= mxReset, 
	mxEmergency:= mxEmergency[4] OR mxEmergency[5] OR mxEmergency[6], 
	mxAutoMode:= mxAutoMode, 
	mxFirstCycle:= mxFirstCycle,
	mrModPosConveyor:= OutfeedConveyor.mrActModPos, 
	mxDisableCollision:= mxHMI_DisableCollision,
	MachParameters:= MachParameters.GantryB, 
	ProdParameters:= ProdParameters.GantryB, 
	SysParameters:= SysParameters.GantryB,
	mxProductPickedUp=> mxProductPickedUpGantry_B,
	Errors=> Errors.Gantry_B);
	
OutfeedConveyor(
	mxReset:= mxReset, 
	mxEmergency:= mxEmergency[6] OR mxEmergency[7], 
	mxAutoMode:= mxAutoMode, 
	mxFirstCycle:= mxFirstCycle,
	MachParameters:= MachParameters.OutfeedConveyor, 
	ProdParameters:= ProdParameters.OutfeedConveyor, 
	SysParameters:= SysParameters.OutfeedConveyor,
	Errors=> Errors.OutfeedConveyor);
	
mxGantrysNotBusy:= NOT GantryA.mxCycleBusy AND NOT GantryB.mxCycleBusy;
END_ACTION

END_FUNCTION_BLOCK

// ---- POUs/ProductHandling/FB_Gantry.TcPOU
FUNCTION_BLOCK FB_Gantry
VAR CONSTANT
	sCycleStateTextDef: ARRAY[0..10]  OF STRING :=	
		['State 0: Wait for Start','1','2','3','4','5','6','7','8','9',
		'State 10: Error'];
	
	tCycleStateTimeouts: ARRAY[0..10] OF TIME := 
		[T#10S,T#10S,T#10S,T#10S,T#10S,T#10S,T#10S,T#10S,T#10S,T#10S,
		T#10S];

	sInitStateTextDef: ARRAY[0..10] OF STRING :=
		['State 0: Wait for Start',
		'State 1: Description Init State 1',
		'State 2: Description Init State 2',
		'State 3; Description Init State 3',
		'State 4; Description Init State 4',
		'State 5; Description Init State 5',
		'State 6; Error State'];

	tInitStateTimeouts: ARRAY[0..10] OF TIME := 
		[T#10S,T#10S,T#10S,T#10S,T#10S,T#10S,T#10S,T#10S,T#10S,T#10S
		,T#10S];
END_VAR
VAR_INPUT
	mxResetCycleState				: BOOL;
	mxResetInitState				: BOOL;
	mxForceInit						: BOOL; (*Reset Calibration Flag*)
	mxReset							: BOOL;	(*Reset Error*)
	mxEmergency						: BOOL;
	mxAutoMode						: BOOL; (* TRUE = Automode *)
	mxFirstCycle					: BOOL;

	mrModPosConveyor				: LREAL;
	mxProductReadyAtTakeout			: BOOL; (* Signal from BottomMold, Takeout Unit *)
	mxDisableCollision				: BOOL;
END_VAR
VAR_IN_OUT
	MachParameters					: ST_GantryMachPar;
	ProdParameters					: ST_GantryProdPar;
	SysParameters					: ST_GantrySysPar;
END_VAR
VAR_OUTPUT
	(*Errors*)
	Errors							: ST_GantryErrors;
	mxErrorInit						: BOOL;		(* Error, stop immediately. Initialisation neccesary *)
	mxErrorStopinPos				: BOOL;		(* Error, stop in position. Only reset neccesary *)

(* State vars *)
	mxCycleBusy						: BOOL;
	mxInitBusy						: BOOL;
	
(* Vars *)
	mxInitialized					: BOOL;
	mrActPosHorizontal				: LREAL;
	mrActPosVertical				: LREAL;
	mxHorizontalIsMoving			: BOOL;
	mxVerticalIsMoving				: BOOL;
	
	(* Signals *)
	mxIsEmpty						: BOOL;
	mxProductPickedUp				: BOOL;
END_VAR
VAR
(* State vars *)
	miCycleState					: INT :=0;
	miCycleOldstate					: INT :=0;
	mxCycleTransitionState			: BOOL := FALSE;
	sCycleStateText					: STRING;
	exCycleTimeOut					: BOOL;		(* Timeout for the whole programcycle *)
	CycleTimeout					: TON;
	CycleTimeOutUpFlank				: R_TRIG;
	mxCycleTimeoutEnable			: BOOL;
	CycleTime						: REAL;
	mxCycleHasError					: BOOL;
	miStopState						: INT;
	mxStartCycle					: BOOL;
	mxStopCycle						: BOOL;
	mxStopDirect					: BOOL;
	
	miInitState						: INT	:=0;
	miInitOldstate					: INT	:=0;
	mxInitTransitionState			: BOOL	:= FALSE;
	sInitStateText					: STRING;
	exInitTimeOut					: BOOL;		(* Timeout for the whole programcycle *)
	InitTimeout						: TON;
	InitTimeOutUpFlank				: R_TRIG;
	mxInitTimeoutEnable				: BOOL;
	InitTime						: REAL;
	mxInitHasError					: BOOL;
	mxStartInit						: BOOL;
	mxStopInit						: BOOL;

	ixCollision						AT %I*: BOOL;	(* Vertical axis *)
	ixEndLimitHorFront				AT %I*: BOOL;
	ixEndLimitHorBack				AT %I*: BOOL;
	ixEndLimitVertUp				AT %I*: BOOL;
	ixEndLimitVertDown				AT %I*: BOOL;
	
	(* Objects *)
	HorizontalAxis					: FB_NcAxis;
	VerticalAxis					: FB_NcAxis;
	(* Pickup Head *)
	BlowOff							: ARRAY [1..6] OF FB_MonoValveNoFdbck;
	VacuumValve						: ARRAY [1..6] OF FB_MonoValveNoFdbck;
	ixVacuumSensor					 AT %I* : ARRAY [1..6] OF BOOL;

(* Vars *)	
	miVacSection					: INT;
	miBlowOffSection				: INT;
	
	mxSwitchVacuumOn				: BOOL;
	(* Errors *)
	SR_exCollision					: SR;
	SR_exEndLimitHorFront			: SR;
	SR_exEndLimitHorBack			: SR;
	SR_exEndLimitVertUp				: SR;
	SR_exEndLimitVertDown			: SR;
	SR_exProductLost				: ARRAY [1..6] OF SR;
	T_VacSensor						: ARRAY [1..6] OF TON;
	mxSwitchBlowOffOn				: BOOL;
	T_WaitAtPickupPosition: TON;
	RT_DropOffPosCoveyor: R_TRIG;
	T_BlowOff: TON;
	mxTemp: BOOL;
	mxTemp2: BOOL;
	mxTest: BOOL;
	FT_SwitchVacuumOff: F_TRIG;
	FT_SwitchBlowOff: F_TRIG;
END_VAR

Error();
Cycle();
Init();
Objects();

ACTION Cycle:
(*StateChange (Transition)  Signalgeneration*)
mxCycleTransitionState:=(miCycleState<>miCycleOldstate);
(*State text*)
sCycleStateText:=sCycleStateTextDef[miCycleState];
(*Timeout Watchdog for Statemachine*)
mxCycleTimeoutEnable:=NOT (miCycleState=0) AND NOT mxReset;

CycleTimeout(IN:=mxCycleTimeoutEnable, PT:=tCycleStateTimeouts[miCycleState] );
CycleTimeOutUpFlank(CLK:=CycleTimeout.Q );
miCycleOldstate:=miCycleState;

(*Set Errorbit when Raising edge of Timeout has been detected*)
IF CycleTimeOutUpFlank.Q THEN
	exCycleTimeOut:=TRUE; 			(* 1 Timeout for the whole programcycle *)
END_IF

(*Function to reset the Statemachine*)
IF mxResetCycleState THEN
	mxResetCycleState:= FALSE;
	miCycleState:=0;
	miCycleOldstate:=miCycleState;
	mxCycleTransitionState:=FALSE;

	mxInitialized:= FALSE;
	mxStartCycle:= FALSE;
	mxStopCycle:= FALSE;
	mxStopDirect:= FALSE;

	mxIsEmpty:= FALSE;
	mxProductPickedUp:= FALSE;
	mxSwitchBlowOffOn:= FALSE;
	mxSwitchVacuumOn:= FALSE;

	T_WaitAtPickupPosition.IN:= FALSE;
	T_BlowOff.IN:= FALSE;
END_IF

fT_SwitchVacuumOff(CLK:= mxSwitchVacuumOn);
FT_SwitchBlowOff(CLK:=mxSwitchBlowOffOn);


(*Definition State has Error*)
mxCycleHasError:=FALSE;

// Open active valves on switch vacuum on.
IF (mxSwitchVacuumOn AND mxAutoMode) THEN
	IF MachParameters.EnableVacuumSection[1] THEN VacuumValve[1].M_On(); END_IF
	IF MachParameters.EnableVacuumSection[2] THEN VacuumValve[2].M_On(); END_IF
	IF MachParameters.EnableVacuumSection[3] THEN VacuumValve[3].M_On(); END_IF
	IF MachParameters.EnableVacuumSection[4] THEN VacuumValve[4].M_On(); END_IF
END_IF

// On trigger, close active valves
IF fT_SwitchVacuumOff.q AND mxAutoMode THEN
	IF MachParameters.EnableVacuumSection[1] THEN VacuumValve[1].M_Off(); END_IF
	IF MachParameters.EnableVacuumSection[2] THEN VacuumValve[2].M_Off(); END_IF
	IF MachParameters.EnableVacuumSection[3] THEN VacuumValve[3].M_Off(); END_IF
	IF MachParameters.EnableVacuumSection[4] THEN VacuumValve[4].M_Off(); END_IF
END_IF

// Open blowoff valves
IF mxSwitchBlowOffOn AND mxAutoMode THEN
	BlowOff[1].M_On();
	BlowOff[2].M_On();
	BlowOff[3].M_On();
	BlowOff[4].M_On();
END_IF

// On trigger, close blowoff valves.
IF FT_SwitchBlowOff.q AND mxAutoMode THEN
	BlowOff[1].M_Off();
	BlowOff[2].M_Off();
	BlowOff[3].M_Off();
	BlowOff[4].M_Off();
END_IF

RT_DropOffPosCoveyor(CLK:= mrModPosConveyor > MachParameters.DropOffConveyorPostion);
T_WaitAtPickupPosition(IN:= , PT:= T#1S);		
T_BlowOff(IN:= , PT:= ProdParameters.BlowOffTime);
IF T_BlowOff.Q THEN T_BlowOff.IN:= FALSE; END_IF
	
(*Cycle State's*)
CASE miCycleState OF
	0:
	(*
	
	- StopCyle en mxPause -> stop bewegingen.
	- Stop Cycle -> empty machine, ga naar rust
	
		- wait for startcycle
		- wait for product ready at takeout
		- Move horizontal to product pickup
		- move vertical to product pickup
		- Vacuum on
		- Move vertical up to transport pos
		- Move horizontal to drop off position (Rest)
		- wait for drop off position conveyor
		- Move vertical down to dropoff position
		- Blow off product
		- Move vertical up to transport pos
		- Goto 1

		* During vertical down, guard the collission sensor=> stop hor and vertical
		* Vacuum sensor check when vacuum on=> error leakage
		*  
	*)
		IF mxStartCycle THEN
			mxStartCycle:= FALSE;
			mxIsEmpty:= FALSE;
			mxProductPickedUp:= FALSE;

			miCycleState:= 1;
		END_IF	

	(* Set when goto 1 mxIsEmpty:= FALSE;	*)

	(* Wait for product ready at takeout *)
	1:
		IF mxStopDirect THEN
			mxStopDirect:= FALSE;
			
			miCycleState:= 25;
		//ELSIF mxStopCycle AND mxPause THEN
		//	mxPause:= FALSE;
			
		//	miCycleState:= 0;
		ELSIF mxStopCycle THEN
			mxStopCycle:= FALSE;
			VerticalAxis.M_Stop();
			HorizontalAxis.M_Stop();
			
			miStopState:= miCycleState;
			miCycleState:= 20;
		ELSIF mxProductReadyAtTakeout THEN
			mxProductReadyAtTakeout:= FALSE;
			mxIsEmpty:= FALSE;
			mxProductPickedUp:= FALSE;
			
			miCycleState:= 2;
		END_IF
		
	(* Move horizontal to the front to pickup position *)
	2:
		IF mxStopDirect THEN
			mxStopDirect:= FALSE;
			
			miCycleState:= 25;
		ELSIF mxStopCycle THEN
			mxStopCycle:= FALSE;
			VerticalAxis.M_Stop();
			HorizontalAxis.M_Stop();
			
			miStopState:= miCycleState;
			miCycleState:= 20;
		ELSIF HorizontalAxis.M_MoveAbsolute(Position:= MachParameters.PositionHorizontalPickup, Velocity:= MachParameters.Hor_VelocityAuto) THEN

			mxSwitchVacuumOn:= TRUE;
			
			miCycleState:=3;
		END_IF

	(* Move Vertical down to pickup position, vacuum on *)
	3:
		IF mxStopDirect THEN
			mxStopDirect:= FALSE;
			
			miCycleState:= 25;
		ELSIF mxStopCycle THEN
			mxStopCycle:= FALSE;
			
			miStopState:= miCycleState;
			miCycleState:= 20;
		ELSIF VerticalAxis.M_MoveAbsolute(Position:= ProdParameters.PositionVerticalPickup, Velocity:= MachParameters.Vert_VelocityAuto) THEN
		
			miCycleState:= 4;
		END_IF

	(* Wait at pickup position *)	
	4:
		T_WaitAtPickupPosition.IN:= TRUE;
	
		IF mxStopDirect THEN
			mxStopDirect:= FALSE;
			
			miCycleState:= 25;
		ELSIF mxStopCycle THEN
			mxStopCycle:= FALSE;
			
			miStopState:= miCycleState;
			miCycleState:= 20;
		ELSIF T_WaitAtPickupPosition.Q THEN
			T_WaitAtPickupPosition.IN:= FALSE;
			
			miCycleState:= 5;
		END_IF		

	(* Move Vertical up to transport position *)
	5:
		IF mxStopDirect THEN
			mxStopDirect:= FALSE;
			
			miCycleState:= 25;
		ELSIF mxStopCycle THEN
			mxStopCycle:= FALSE;
			
			miStopState:= miCycleState;
			miCycleState:= 20;
		ELSIF VerticalAxis.M_MoveAbsolute(Position:= MachParameters.Vert_PositionTransport, Velocity:= MachParameters.Vert_VelocityAuto) THEN
			mxProductPickedUp:= TRUE;

			miCycleState:= 6;
		END_IF
		
	(* Move horizontal to the back to drop-off position *)
	6:
		IF mxStopDirect THEN
			mxStopDirect:= FALSE;
			
			miCycleState:= 25;
		ELSIF mxStopCycle THEN
			mxStopCycle:= FALSE;
			
			miStopState:= miCycleState;
			miCycleState:= 20;
		ELSIF HorizontalAxis.M_MoveAbsolute(Position:= MachParameters.PositionHorizontalDropOff, Velocity:= MachParameters.Hor_VelocityAuto) THEN
			mxProductPickedUp := FALSE;
			miCycleState:= 7;
		END_IF
		
	(* Wait for drop off position conveyor *)
	7:
		IF mxStopDirect THEN
			mxStopDirect:= FALSE;
			
			miCycleState:= 25;
		ELSIF mxStopCycle THEN
			mxStopCycle:= FALSE;
			
			miStopState:= miCycleState;
			miCycleState:= 20;
		ELSIF RT_DropOffPosCoveyor.Q THEN
			
			miCycleState:= 8;
		END_IF

	(* Move Vertical Axis down to drop off position *)
	8:
		IF mxStopDirect THEN
			mxStopDirect:= FALSE;
			
			miCycleState:= 25;
		ELSIF mxStopCycle THEN
			mxStopCycle:= FALSE;
			
			miStopState:= miCycleState;
			miCycleState:= 20;
		ELSIF VerticalAxis.M_MoveAbsolute(Position:= ProdParameters.PositionVerticalDropOff, Velocity:= MachParameters.Vert_VelocityAuto) THEN
			T_BlowOff.IN:= TRUE;
			mxSwitchBlowOffOn := TRUE;
			mxSwitchVacuumOn := FALSE; // bateu 20180619
			
			miCycleState:= 9;
		END_IF
		
	(* Move Vertical Axis up to transport position *)
	9:
		IF mxStopDirect THEN
			mxStopDirect:= FALSE;
			
			miCycleState:= 25;
		ELSIF mxStopCycle THEN
			mxStopCycle:= FALSE;
			
			miStopState:= miCycleState;
			miCycleState:= 20;
		ELSIF T_BlowOff.q THEN
			T_BlowOff.IN := FALSE;
			mxSwitchBlowOffOn := FALSE;
			miCycleState:= 10;
		END_IF
	
	10:
		IF mxStopDirect THEN
			mxStopDirect:= FALSE;
			
			miCycleState:= 25;
		ELSIF mxStopCycle THEN
			mxStopCycle:= FALSE;
			
			miStopState:= miCycleState;
			miCycleState:= 20;
		ELSIF VerticalAxis.M_MoveAbsolute(Position:= MachParameters.Vert_PositionTransport, Velocity:= MachParameters.Vert_VelocityAuto) THEN
			//mxIsEmpty:= TRUE;
			
			miCycleState:= 11;
		END_IF

	(* Move Horizontal Axis to rest position *)
	11:
		IF mxStopDirect THEN
			mxStopDirect:= FALSE;
			
			miCycleState:= 25;
		ELSIF mxStopCycle THEN
			mxStopCycle:= FALSE;
			
			miStopState:= miCycleState;
			miCycleState:= 20;
		ELSIF HorizontalAxis.M_MoveAbsolute(Position:= MachParameters.Hor_Positionrest, Velocity:= MachParameters.Hor_VelocityAuto) THEN
			mxIsEmpty:= TRUE;
			
			miCycleState:= 1;
		END_IF

	(* Stop Cycle *)
	20:
		IF mxStopDirect THEN
			mxStopDirect:= FALSE;
			
			miCycleState:= 21;
		ELSE 
			VerticalAxis.M_Stop();
			HorizontalAxis.M_Stop();
			
			miCycleState:= 21;
		END_IF
	
	(* Stop Cycle, wait for gantry's stopped *)
	21:
		IF mxStopDirect THEN
			mxStopDirect:= FALSE;
			
			miCycleState:= 21;
		ELSIF (HorizontalAxis.axStatus.StandStill OR NOT HorizontalAxis.axStatus.Moving) AND (VerticalAxis.axStatus.StandStill OR NOT VerticalAxis.axStatus.Moving) THEN
			
			miCycleState:= 22;
		END_IF

	(* Stop Cycle, wait for restart *)
	22:
		IF mxStopDirect THEN
			mxStopDirect:= FALSE;
			
			miCycleState:= 21;
		ELSIF mxStartCycle THEN
			mxStartCycle:= FALSE;
			
			miCycleState:= miStopState;
		END_IF

	(* Stop Direct *)
	25:
		mxInitialized:= FALSE;
		mxStartCycle:= FALSE;
		mxStopCycle:= FALSE;
		mxStopDirect:= FALSE;

		mxIsEmpty:= FALSE;
		mxProductPickedUp:= FALSE;
		mxSwitchBlowOffOn:= FALSE;
		mxSwitchVacuumOn:= FALSE;

		T_WaitAtPickupPosition.IN:= FALSE;
		T_BlowOff.IN:= FALSE;

		miCycleState:= 0;
END_CASE

mxCycleBusy:= miCycleState<>0 AND NOT (miCycleState=22);
END_ACTION

ACTION Error:
SR_exCollision(SET1:= NOT ixCollision AND NOT mxDisableCollision, RESET:= mxReset, Q1=> Errors.Collision);
SR_exEndLimitHorFront(SET1:= NOT ixEndLimitHorFront, RESET:= mxReset, Q1=> Errors.EndLimitHorFront);
SR_exEndLimitHorBack(SET1:= NOT ixEndLimitHorBack, RESET:= mxReset, Q1=> Errors.EndLimitHorBack);
SR_exEndLimitVertUp(SET1:= NOT ixEndLimitVertUp, RESET:= mxReset, Q1=> Errors.EndLimitVertUp);
SR_exEndLimitVertDown(SET1:= NOT ixEndLimitVertDown, RESET:= mxReset, Q1=> Errors.EndLimitVertDown);

(*
FOR miVacSection:= 1 TO 6 DO
T_VacSensor[miVacSection](IN:= VacuumValve[miVacSection].mxIsOn, PT:= T#3S);
SR_exProductLost[miVacSection](
		SET1:= MachParameters.EnableVacuumSection[miVacSection] AND VacuumValve[miVacSection].mxIsOn AND (T_VacSensor[miVacSection].Q AND NOT ixVacuumSensor[miVacSection]) , 
		RESET:= mxReset, Q1=> Errors.ProductLost[miVacSection]);
END_FOR
*)

T_VacSensor[1](IN:= VacuumValve[1].mxIsOn, PT:= T#3S);
SR_exProductLost[1](
		SET1:= MachParameters.EnableVacuumSection[1] AND VacuumValve[1].mxIsOn AND (T_VacSensor[1].Q AND NOT ixVacuumSensor[1]) , 
		RESET:= mxReset, Q1=> Errors.ProductLost[1]);
		
T_VacSensor[2](IN:= VacuumValve[2].mxIsOn, PT:= T#3S);
SR_exProductLost[2](
		SET1:= MachParameters.EnableVacuumSection[2] AND VacuumValve[2].mxIsOn AND (T_VacSensor[2].Q AND NOT ixVacuumSensor[2]) , 
		RESET:= mxReset, Q1=> Errors.ProductLost[2]);
		
T_VacSensor[3](IN:= VacuumValve[3].mxIsOn, PT:= T#3S);
SR_exProductLost[3](
		SET1:= MachParameters.EnableVacuumSection[3] AND VacuumValve[3].mxIsOn AND (T_VacSensor[3].Q AND NOT ixVacuumSensor[3]) , 
		RESET:= mxReset, Q1=> Errors.ProductLost[3]);
		
T_VacSensor[4](IN:= VacuumValve[4].mxIsOn, PT:= T#3S);
SR_exProductLost[4](
		SET1:= MachParameters.EnableVacuumSection[4] AND VacuumValve[4].mxIsOn AND (T_VacSensor[4].Q AND NOT ixVacuumSensor[4]) , 
		RESET:= mxReset, Q1=> Errors.ProductLost[4]);






(*************************************************************************************************)
mxErrorInit:= Errors.Collision OR Errors.EndLimitHorFront OR Errors.EndLimitHorBack OR Errors.EndLimitVertUp OR Errors.EndLimitVertDown OR
	HorizontalAxis.ErrorStop OR VerticalAxis.ErrorStop;;
mxErrorStopinPos:= FALSE;
END_ACTION

ACTION Init:
(*StateChange (Transition)  Signalgeneration*)
mxInitTransitionState:=(miInitState<>miInitOldstate);
(*State text*)
sInitStateText:=sInitStateTextDef[miInitState];
(*Timeout Watchdog for Statemachine*)
mxInitTimeoutEnable:=NOT (miInitState=0)  AND NOT mxReset;

InitTimeout(IN:=mxInitTimeoutEnable  , PT:=tInitStateTimeouts[miInitState] );
InitTimeOutUpFlank(CLK:=InitTimeout.Q );
miInitOldstate:=miInitState;

(*Set Errorbit when Raising edge of Timeout has been detected*)
IF InitTimeOutUpFlank.Q THEN
	exInitTimeOut:=TRUE; 			(* 1 Timeout for the whole programcycle *)
END_IF

(*Function to reset the Statemachine*)
IF mxResetInitState THEN
	mxResetInitState:=FALSE;
	miInitState:=0;
	miInitOldstate:=miInitState;
	mxInitTransitionState:=FALSE;

	mxInitialized:= FALSE;	
	mxStartInit:= FALSE;
	mxStopInit:= FALSE;
END_IF

(*Definition State has Error*)
mxInitHasError:=FALSE;

(*Init State's*)
CASE miInitState OF
	0:
	
	(* 
		- Wait for start int
		- Blow off uit
		- vacuum aan laten
		- Vertical move up to transport pos.
		- Horizontal move back to drop off positie
		- 	
	
	*)
		IF mxStartInit THEN
			mxStartInit:= FALSE;
			mxInitialized:= FALSE;

			(* Don't turn vacuum off, turn blowoff off *)
			mxSwitchBlowOffOn:= FALSE;
			
			miInitState:= 1;
		END_IF

	(* Move vertical up *)
	1:
		IF mxStopInit THEN
			mxStopInit:= FALSE;
			
			miInitState:= 10;
		ELSIF VerticalAxis.M_MoveAbsolute(Position:= MachParameters.Vert_PositionTransport, Velocity:= MachParameters.Vert_VelocityAuto) THEN
			
			miInitState:= 2;			
		END_IF

	(* Move horizontal back *)
	2:
		IF mxStopInit THEN
			mxStopInit:= FALSE;

			miInitState:= 10;
		ELSIF HorizontalAxis.M_MoveAbsolute(Position:= MachParameters.Hor_Positionrest, Velocity:= MachParameters.Hor_VelocityAuto) THEN
			
			mxInitialized:= TRUE;
			miInitState:= 0;			
		END_IF

	(* Stop Init *)
	10:
		mxInitialized:= FALSE;	
		mxStartInit:= FALSE;
		mxStopInit:= FALSE;

		VerticalAxis.M_Stop();
		HorizontalAxis.M_Stop();
		
		miInitState:= 0;
		
END_CASE

mxInitBusy:= miInitState<>0;
END_ACTION

METHOD M_StartCycle

IF NOT mxCycleBusy THEN
	mxStartCycle:= TRUE;	
END_IF
END_METHOD

METHOD M_StartInit
VAR_INPUT
END_VAR

IF NOT mxInitBusy THEN
	mxStartInit:= TRUE;
END_IF
END_METHOD

METHOD M_StopCycle

IF mxCycleBusy THEN 
	mxStopCycle:= TRUE; 
END_IF
END_METHOD

METHOD M_StopDirect

IF mxCycleBusy THEN
	mxStopDirect:= TRUE;	
END_IF
END_METHOD

METHOD M_StopInit

IF mxInitBusy THEN 
	mxStopInit:= TRUE; 
END_IF
END_METHOD

ACTION Objects:
HorizontalAxis(
	mxEnable:= NOT mxEmergency, 
	mxInhibit:= FALSE, 
	mxAutoMode:= mxAutoMode, 
	mxReset:= mxReset, 
	mxFirstCycle:= 	mxFirstCycle,
	mxEmergency:= mxEmergency, 
	mxSimulation:= , 
	mxResetCycle:= , 
	mxDisable_Positive:= NOT ixEndLimitHorFront, 
	mxDisable_Negative:= NOT ixEndLimitHorBack, 
	mxBlockHMI:= , 
	mrOverride:= 100.0,
	mrVelocityManual:= MachParameters.Hor_VelocityManual,
	mrHomePos:= MachParameters.Hor_PositionHome, 
	SysParameters:= SysParameters.HorizontalAxis,
	mxCycleBusy=> , 
	mxRunning=> , 
	Errors=> Errors.HorizontalNCAxisError, 
	Error=> , 
	ErrorStop=> , 
	axStatus=> , 
	mxAxisIsMoving=> mxHorizontalIsMoving,
	ActPosition=> mrActPosHorizontal, 
	ActVelocity=> , 
	axAxis=> );
	
VerticalAxis(
	mxEnable:= NOT mxEmergency, 
	mxInhibit:= FALSE, 
	mxAutoMode:= mxAutoMode, 
	mxReset:= mxReset, 
	mxFirstCycle:= 	mxFirstCycle,
	mxEmergency:= mxEmergency, 
	mxSimulation:= , 
	mxResetCycle:= , 
	mxDisable_Positive:= NOT ixEndLimitVertUp, 
	mxDisable_Negative:= (NOT ixEndLimitVertDown) OR Errors.Collision, 
	mxBlockHMI:= , 
	mrOverride:= 100.0, 
	mrVelocityManual:= MachParameters.Vert_VelocityManual, 
	mrHomePos:= MachParameters.Vert_PositionHome, 
	SysParameters:= SysParameters.VerticalAxis,
	mxCycleBusy=> , 
	mxRunning=> , 
	Errors=> Errors.VerticalNCAxisError, 
	Error=> , 
	ErrorStop=> , 
	axStatus=> , 
	mxAxisIsMoving=> mxVerticalIsMoving,
	ActPosition=> mrActPosVertical, 
	ActVelocity=> , 
	axAxis=> );

FOR miVacSection:= 1 TO 6 DO	
	VacuumValve[miVacSection](
		mxReset:= mxReset, 
		mxEmergency:= mxEmergency, 
		mxAutoMode:= mxAutoMode, 
		mxIsOn=> );
END_FOR
FOR miBlowOffSection:= 1 TO 6 DO
	BlowOff[miBlowOffSection](
		mxReset:= mxReset, 
		mxEmergency:= mxEmergency, 
		mxAutoMode:= mxAutoMode, 
		mxIsOn=> );
END_FOR
END_ACTION

END_FUNCTION_BLOCK

// ---- POUs/Standard/FB_Blink.TcPOU
FUNCTION_BLOCK FB_Blink
VAR_INPUT
END_VAR
VAR_OUTPUT
	Fast:BOOL;
	Normal:BOOL;
	Slow:BOOL;
END_VAR
VAR
	TFast:TON;
	TNormal:TON;
	TSlow:TON;

END_VAR

TFast(IN:=NOT TFast.Q , PT:=T#0.1S);
TNormal(IN:=NOT TNormal.Q , PT:=T#0.2S);
TSlow(IN:=NOT TSlow.Q , PT:=T#0.3S);

IF TFast.Q THEN
	(*Toggle bit*)
	Fast:=NOT Fast;
END_IF

IF TNormal.Q THEN
	(*Toggle bit*)
	Normal:=NOT Normal;
END_IF

IF TSlow.Q THEN
	(*Toggle bit*)
	Slow:=NOT Slow;
END_IF

END_FUNCTION_BLOCK

// ---- POUs/Standard/GateRequest.TcPOU
(******************************************************************************)
(*	Gate request															  *)
(******************************************************************************)
FUNCTION_BLOCK GateRequest
VAR_INPUT
	GateClosed 			: BOOL; (* Gate closed signal(s) from safety program *)
	SafeState			: BOOL; (* Machine is in safe state *)
	Request_Open 		: BOOL; (* Request door open *)
	Reset				: BOOL; (* Reset Button from safety program *)
	TimeOutSafeState	: TIME:= T#5S; (* Max time for safe state *)
END_VAR
VAR_OUTPUT
	Lock 				: BOOL; (* Activate lock(s) *)
	GateRequest_Light 	: BOOL; (* Light request button *)
	ResetButton_Light 	: BOOL; (* Light reset button *)
END_VAR
VAR
	TimerFlashOn		: TON; (* Timer for flash on *)
	TimerFlashOff		: TON; (* Timer for Flash off *)
	Flash				: SR; (* Flash function *)
END_VAR

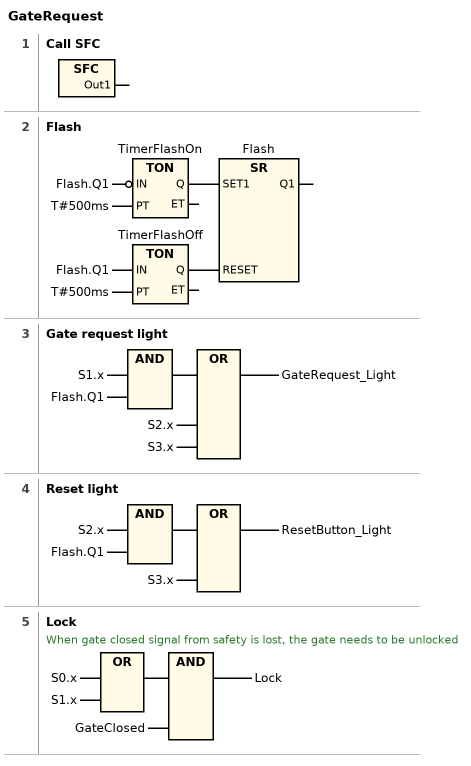
// NETWORK 1: Call SFC
SFC();

// NETWORK 2: Flash
TimerFlashOn(IN := NOT Flash.Q1, PT := T#500ms); // TON
TimerFlashOff(IN := Flash.Q1, PT := T#500ms); // TON
Flash(SET1 := TimerFlashOn.Q, RESET := TimerFlashOff.Q); // SR

// NETWORK 3: Gate request light
GateRequest_Light := S1.x AND Flash.Q1 OR S2.x OR S3.x;

// NETWORK 4: Reset light
ResetButton_Light := S2.x AND Flash.Q1 OR S3.x;

// NETWORK 5: Lock
// When gate closed signal from safety is lost, the gate needs to be unlocked
Lock := (S0.x OR S1.x) AND GateClosed;

ACTION SFC:
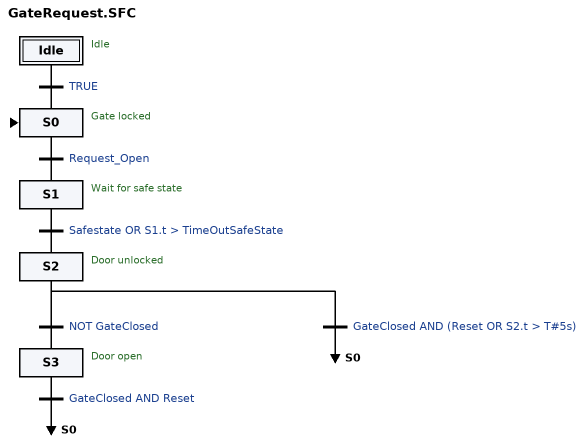
// Idle
INITIAL_STEP Idle:
END_STEP
TRANSITION FROM Idle TO S0
    := TRUE;
END_TRANSITION
// Gate locked
STEP S0:
END_STEP
TRANSITION FROM S0 TO S1
    := Request_Open;
END_TRANSITION
// Wait for safe state
STEP S1:
END_STEP
TRANSITION FROM S1 TO S2
    := Safestate OR S1.t > TimeOutSafeState;
END_TRANSITION
// Door unlocked
STEP S2:
END_STEP
TRANSITION FROM S2 TO S3
    := NOT GateClosed;
END_TRANSITION
TRANSITION FROM S2 TO S0
    := GateClosed AND (Reset OR S2.t > T#5s);
END_TRANSITION
// Door open
STEP S3:
END_STEP
TRANSITION FROM S3 TO S0
    := GateClosed AND Reset;
END_TRANSITION
END_ACTION

END_FUNCTION_BLOCK

// ---- POUs/Standard/FB_EthercatDiag.TcPOU
FUNCTION_BLOCK FB_EtherCATDiag
VAR_INPUT
(* EtherCAT *)
	SlaveCount 		:UINT;		(* Actual count of EtherCAT slaves received *)
	CfgSlaveCount	:UINT;		(* Count of configured EtherCAT slaves *)

	DevState 		:UINT;		(* EtherCAT State:
									0x0001 = Link error
									0x0002 = I/O locked after link error (I/O reset required)
									0x0004 = Link error (redundancy adapter)
									0x0008 = Missing one frame (redundancy mode)
									0x0010 = Out of send resources (I/O reset required)
									0x0020 = Watchdog triggered
									0x0040 = Ethernet driver (miniport) not found
									0x0080 = I/O reset active
									0x0100 = At least one device in 'INIT' state
									0x0200 = At least one device in 'PRE-OP' state
									0x0400 = At least one device in 'SAFE-OP' state
									0x0800 = At least one device indicates an error state
									0x1000 = DC not in sync
								 *)
END_VAR

VAR_OUTPUT
(* Alarms*)
	EtherCATLinkError			: BOOL;		(* EtherCAT error, link error *)
	EtherCATSlaveMissing		: BOOL;		(* EtherCAT error, at least one device not connected *)
	EtherCATOPmode				: BOOL;		(* EtherCAT error, at leat one device not in 'OP'-mode *)
	EtherCATResetNeeded			: BOOL;		(* EtherCAT error, I/O reset required *)
END_VAR

VAR
	Fx: WORD;

	bInit						: BOOL;		(* At least one device in 'INIT' state *)
	bPreOP						: BOOL;		(* At least one device in 'PRE-OP' state *)
	bSafeOP						: BOOL;		(* At least one device in 'SAFE-OP' state *)
	bError						: BOOL;		(* At least one device indicates an error state *)
	bIOLocked					: BOOL;		(* I/O locked after link error (I/O reset required) *)
	bNoResources				: BOOL;		(* Out of send resources (I/O reset required) *)
END_VAR

(*----------------------------------------------------------------------------------------------------------------*)
(* Slave missing form EtherCAT bus *)
(* Alarm message: EtherCAT error, at least one device not connected *)
IF SlaveCount <> CfgSlaveCount
THEN
	EtherCATSlaveMissing	:= TRUE;
ELSE
	EtherCATSlaveMissing	:= FALSE;
END_IF


(*----------------------------------------------------------------------------------------------------------------*)
(* EtherCAT device link error *)
Fx := UINT_TO_WORD(DevState) AND 16#0001;

IF Fx = 16#0001
THEN
	EtherCATLinkError := TRUE;
ELSE
	EtherCATLinkError := FALSE;
END_IF


(*----------------------------------------------------------------------------------------------------------------*)
(* EtherCAT device not in 'OP'-mode *)
(* Check devices for INIT-state *)
Fx	:= UINT_TO_WORD( DevState ) AND 16#0100;

IF Fx = 16#0100
THEN
	bInit		:= TRUE;
ELSE
	bInit 		:= FALSE;
END_IF

(* Check devices for PREOP-state *)
Fx := UINT_TO_WORD( DevState ) AND 16#0200;

IF Fx = 16#0200
THEN
	bPreOP		:= TRUE;
ELSE
	bPreOP 		:= FALSE;
END_IF

(* Check devices for SAFEEOP-state *)
Fx := UINT_TO_WORD( DevState ) AND 16#0400;

IF Fx = 16#0400
THEN
	bSafeOP		:= TRUE;
ELSE
	bSafeOP 	:= FALSE;
END_IF

(* Check devices for error-state *)
Fx := UINT_TO_WORD( DevState ) AND 16#0800;

IF Fx = 16#0800
THEN
	bError		:= TRUE;
ELSE
	bError 		:= FALSE;
END_IF

(* At least one device not in OP-mode *)
EtherCATOPmode	:=			bInit
						OR	bPreOP
						OR	bSafeOP
						OR	bError;


(*----------------------------------------------------------------------------------------------------------------*)
(* EtherCAT I/O reset needed *)
(* Check for any I/O lock *)
Fx := UINT_TO_WORD( DevState ) AND 16#0002;

IF Fx = 16#0002
THEN
	bIOLocked		:= TRUE;
ELSE
	bIOLocked 		:= FALSE;
END_IF

(* Check for out of send resources *)
Fx := UINT_TO_WORD( DevState ) AND 16#0010;

IF Fx = 16#0010
THEN
	bNoResources		:= TRUE;
ELSE
	bNoResources 		:= FALSE;
END_IF

(* EtherCAT error, I/O reset required *)
EtherCATResetNeeded	:=			bIOLocked
							OR	bNoResources;

END_FUNCTION_BLOCK

// ---- POUs/FB_instancePath.TcPOU
{attribute 'reflection'} 
FUNCTION_BLOCK FB_instancePath 
VAR 
    {attribute 'instance-path'} 
    {attribute 'noinit'} 
    sPath : STRING; 
END_VAR

END_FUNCTION_BLOCK

// ---- POUs/Standard/Analog/FB_AnalogOut0_10V.TcPOU
FUNCTION_BLOCK FB_AnalogOut0_10V
VAR_INPUT
	EngInput				: REAL;
	EngLowLimit				: REAL; (*Low limit*)
	EngUpperLimit 			: REAL; (*Upper limit*)
END_VAR
VAR_OUTPUT
END_VAR
VAR
	VOut 					: REAL;
	RawOut 					AT %Q* : INT;
END_VAR

VOut		:= 10/(EngUpperLimit-EngLowLimit)*(EngInput--EngLowLimit);
RawOut		:= REAL_TO_INT(32767.0/(EngUpperLimit-EngLowLimit)*(EngInput--EngLowLimit));

END_FUNCTION_BLOCK

// ---- POUs/Standard/Balluff/FB_BalluffDevice.TcPOU
FUNCTION_BLOCK FB_BalluffDevice
VAR_INPUT
END_VAR
VAR_OUTPUT
	Error	: BOOL;
	Position: REAL;
	Temperature	: REAL;
END_VAR
VAR
	Device	AT %I* : ST_BalluffDevice;
END_VAR

Error:= (Device.ErrorRegister<>0);
Temperature:= INT_TO_REAL(Device.Temperature);

END_FUNCTION_BLOCK

// ---- POUs/Standard/FIFO/FB_CalculateMaxKO.TcPOU
FUNCTION_BLOCK FB_CalculateMaxKO
VAR_INPUT
	init			: BOOL;
	AEnabled		: BOOL;
	BEnabled		: BOOL;
	Value_A			: REAL;
	Value_B			: REAL;
	Value_Forming	: REAL;
END_VAR
VAR_IN_OUT
	CLK_A 			: BOOL;
	CLK_B 			: BOOL;
	CLK_Forming		: BOOL;
END_VAR
VAR_OUTPUT
	MaxKO			: REAL;
END_VAR
VAR
	MaxKO_Array		: ARRAY [1..6] OF REAL;
	
	RT_CLK_A		: R_TRIG;
	RT_CLK_B		: R_TRIG;
	RT_CLK_Forming	: R_TRIG;
	
